ABB RAPID module: ANV4y1.mod

MODULE ANV4y1

	PERS tooldata Pen:=[TRUE,[[0,0,139],[1,0,0,0]],[0.5,[0,0,20],[1,0,0,0],0,0,0]];
	CONST robtarget origin :=[[0,0,0],[1,0,0,0],[0,0,-1,0],[9E+09,9E+09,9E+09,9E+09,9E+09,9E+09]];
	CONST robtarget home_1:=[[120,148.105008887,-250.933670218],[0.706940789,-0.015320621,0.015320621,0.706940789],[0,0,0,0],[9E+09,9E+09,9E+09,9E+09,9E+09,9E+09]];
	TASK PERS wobjdata paper_obj:=[FALSE,TRUE,"",[[1355,120,401],[0,-0.707106781,0.707106781,0]],[[0,0,0],[1,0,0,0]]];
	VAR num array_x{8510}:= [145,144,144,144,144,144,144,144,144,144,144,144,144,144,144,144,144,144,144,144,144,144,144,144,144,144,144,144,144,144,144,146,146,147,147,148,148,149,149,150,150,151,151,152,152,153,153,154,154,154,154,155,155,156,156,157,157,158,158,159,159,160,160,161,161,162,162,162,162,161,161,160,160,159,159,158,158,157,157,156,156,155,155,154,154,153,153,152,152,151,151,150,150,149,149,149,149,148,148,147,147,146,146,145,145,144,144,143,143,142,142,141,141,140,140,140,140,139,139,138,138,137,137,137,137,136,136,136,136,135,135,135,135,134,134,133,133,133,133,132,132,132,132,131,131,131,131,130,130,130,130,129,129,129,129,128,128,127,127,127,127,126,126,126,126,125,125,125,125,124,124,124,124,123,123,123,123,122,122,122,122,121,121,120,120,120,120,119,119,119,119,118,118,118,118,117,117,117,117,116,116,116,116,115,115,115,115,114,114,113,113,113,113,112,112,112,112,111,111,111,111,111,111,109,109,108,108,107,107,106,106,106,106,105,105,105,105,105,105,105,105,105,105,105,105,105,105,105,105,105,105,105,105,105,105,105,105,105,105,105,105,105,105,105,105,105,105,105,105,105,105,105,105,106,106,106,106,106,106,106,106,106,106,106,106,106,106,106,106,106,106,106,106,106,106,106,106,106,106,106,106,106,106,106,106,106,106,106,106,106,106,106,106,106,106,105,105,105,105,103,103,103,103,104,104,104,104,104,104,104,104,104,104,104,104,104,104,104,104,104,104,104,104,104,104,104,104,104,104,104,104,104,104,104,104,104,104,104,104,104,104,104,104,104,104,103,103,103,103,103,103,103,103,103,103,103,103,103,103,103,103,103,103,103,103,103,103,103,103,103,103,103,103,103,103,103,103,103,103,103,103,103,103,103,103,103,103,101,101,100,100,99,99,98,98,97,97,97,97,97,97,98,98,101,101,102,102,102,102,102,102,101,101,101,101,100,100,99,99,98,98,97,97,98,98,99,99,100,100,101,101,102,102,102,102,102,102,101,101,101,101,100,100,99,99,98,98,98,98,91,91,92,92,93,93,93,93,94,94,95,95,96,96,97,97,97,97,95,95,95,95,95,95,94,94,94,94,93,93,93,93,92,92,92,92,91,91,91,91,90,90,90,90,89,89,89,89,90,90,89,89,89,89,88,88,88,88,87,87,87,87,86,86,86,86,86,86,85,85,84,84,83,83,82,82,82,82,81,81,80,80,79,79,78,78,75,75,75,75,76,76,76,76,77,77,77,77,77,77,78,78,78,78,79,79,79,79,79,79,80,80,80,80,81,81,81,81,81,81,82,82,82,82,83,83,83,83,83,83,84,84,84,84,85,85,85,85,86,86,86,86,86,86,87,87,87,87,87,87,88,88,88,88,88,88,81,81,80,80,80,80,79,79,79,79,79,79,78,78,78,78,77,77,77,77,76,76,76,76,76,76,75,75,75,75,75,75,74,74,74,74,74,74,73,73,73,73,72,72,72,72,71,71,71,71,71,71,70,70,70,70,69,69,69,69,68,68,68,68,68,68,68,68,67,67,67,67,67,67,65,65,65,65,65,65,66,66,66,66,66,66,67,67,67,67,68,68,68,68,69,69,69,69,69,69,70,70,70,70,71,71,71,71,72,72,72,72,73,73,73,73,74,74,74,74,74,74,75,75,76,76,77,77,78,78,81,81,82,82,82,82,83,83,83,83,83,83,84,84,84,84,84,84,85,85,85,85,85,85,86,86,86,86,87,87,87,87,88,88,88,88,88,88,86,86,84,84,84,84,83,83,83,83,82,82,81,81,80,80,79,79,58,58,59,59,59,59,60,60,60,60,60,60,60,60,60,60,60,60,60,60,60,60,60,60,59,59,58,58,57,57,56,56,55,55,54,54,53,53,52,52,51,51,50,50,49,49,48,48,47,47,46,46,45,45,44,44,43,43,42,42,41,41,41,41,40,40,40,40,40,40,40,40,38,38,38,38,37,37,36,36,35,35,34,34,33,33,32,32,31,31,31,31,31,31,32,32,32,32,32,32,33,33,33,33,33,33,34,34,35,35,36,36,36,36,37,37,37,37,37,37,37,37,36,36,39,39,39,39,39,39,38,38,38,38,38,38,37,37,37,37,37,37,32,32,32,32,32,32,32,32,31,31,31,31,31,31,30,30,30,30,30,30,29,29,29,29,29,29,28,28,28,28,28,28,36,36,37,37,38,38,39,39,38,38,38,38,38,38,38,38,38,38,36,36,36,36,36,36,36,36,36,36,37,37,37,37,39,39,39,39,39,39,39,39,37,37,37,37,37,37,39,39,40,40,40,40,40,40,38,38,38,38,38,38,38,38,38,38,39,39,40,40,41,41,53,53,53,53,53,53,53,53,52,52,52,52,52,52,52,52,52,52,52,52,52,52,52,52,52,52,53,53,54,54,54,54,54,54,54,54,54,54,54,54,54,54,54,54,55,55,55,55,55,55,55,55,54,54,53,53,54,54,54,54,54,54,54,54,55,55,55,55,55,55,55,55,55,55,55,55,55,55,55,55,56,56,56,56,56,56,56,56,56,56,56,56,57,57,57,57,57,57,58,58,58,58,61,61,60,60,60,60,60,60,59,59,59,59,59,59,58,58,58,58,58,58,58,58,58,58,58,58,57,57,57,57,57,57,57,57,57,57,57,57,57,57,57,57,56,56,56,56,56,56,56,56,56,56,56,56,64,64,64,64,64,64,63,63,63,63,63,63,62,62,62,62,62,62,61,61,61,61,61,61,61,61,60,60,60,60,60,60,59,59,59,59,59,59,58,58,58,58,58,58,58,58,57,57,57,57,57,57,57,57,57,57,57,57,56,56,53,53,53,53,53,53,53,53,53,53,52,52,51,51,51,51,50,50,50,50,49,49,49,49,48,48,47,47,46,46,45,45,44,44,43,43,43,43,43,43,44,44,45,45,46,46,47,47,48,48,49,49,50,50,51,51,52,52,54,54,54,54,56,56,56,56,56,56,57,57,57,57,58,58,59,59,60,60,61,61,62,62,63,63,63,63,64,64,65,65,67,67,67,67,68,68,69,69,69,69,67,67,67,67,68,68,67,67,68,68,69,69,70,70,71,71,72,72,73,73,74,74,75,75,76,76,77,77,78,78,79,79,80,80,81,81,82,82,83,83,84,84,85,85,86,86,87,87,86,86,85,85,84,84,83,83,82,82,81,81,80,80,79,79,78,78,77,77,76,76,75,75,74,74,73,73,72,72,71,71,70,70,69,69,69,69,69,69,69,69,69,69,69,69,72,72,71,71,71,71,72,72,73,73,74,74,75,75,76,76,77,77,78,78,79,79,80,80,81,81,82,82,83,83,84,84,85,85,86,86,85,85,86,86,87,87,87,87,84,84,83,83,82,82,82,82,81,81,80,80,79,79,79,79,79,79,80,80,81,81,82,82,83,83,84,84,85,85,85,85,86,86,88,88,89,89,89,89,89,89,88,88,87,87,81,81,80,80,79,79,78,78,81,81,81,81,80,80,79,79,78,78,78,78,80,80,80,80,80,80,80,80,79,79,78,78,78,78,78,78,78,78,78,78,78,78,78,78,76,76,76,76,76,76,76,76,76,76,76,76,76,76,76,76,76,76,76,76,77,77,81,81,82,82,83,83,82,82,83,83,84,84,84,84,85,85,86,86,86,86,87,87,86,86,86,86,86,86,87,87,87,87,88,88,89,89,89,89,88,88,89,89,89,89,90,90,108,108,108,108,108,108,108,108,108,108,108,108,108,108,108,108,109,109,109,109,109,109,109,109,109,109,108,108,107,107,106,106,105,105,104,104,103,103,103,103,102,102,101,101,100,100,99,99,98,98,97,97,97,97,96,96,96,96,95,95,94,94,93,93,92,92,91,91,90,90,89,89,88,88,87,87,86,86,85,85,85,85,85,85,86,86,90,90,89,89,89,89,89,89,89,89,90,90,91,91,92,92,92,92,93,93,92,92,91,91,88,88,89,89,90,90,91,91,92,92,93,93,94,94,95,95,96,96,97,97,97,97,98,98,99,99,100,100,100,100,101,101,89,89,87,87,88,88,89,89,89,89,88,88,87,87,86,86,85,85,84,84,82,82,81,81,80,80,79,79,78,78,77,77,76,76,75,75,74,74,73,73,72,72,71,71,70,70,69,69,68,68,67,67,67,67,66,66,66,66,66,66,66,66,67,67,68,68,69,69,69,69,70,70,71,71,72,72,73,73,74,74,75,75,76,76,77,77,78,78,79,79,80,80,81,81,82,82,83,83,83,83,83,83,82,82,81,81,80,80,79,79,78,78,77,77,76,76,75,75,74,74,73,73,72,72,71,71,70,70,69,69,69,69,68,68,68,68,67,67,67,67,70,70,71,71,72,72,73,73,74,74,75,75,76,76,77,77,78,78,79,79,80,80,81,81,81,81,82,82,82,82,82,82,81,81,80,80,79,79,78,78,77,77,76,76,75,75,74,74,73,73,72,72,71,71,70,70,71,71,73,73,70,70,69,69,68,68,67,67,67,67,64,64,64,64,63,63,63,63,63,63,63,63,62,62,61,61,60,60,59,59,59,59,59,59,59,59,59,59,59,59,59,59,60,60,60,60,60,60,60,60,61,61,61,61,61,61,62,62,62,62,62,62,62,62,62,62,63,63,63,63,63,63,64,64,64,64,64,64,64,64,65,65,65,65,65,65,66,66,66,66,66,66,68,68,68,68,69,69,69,69,70,70,70,70,71,71,71,71,72,72,72,72,72,72,73,73,73,73,74,74,74,74,75,75,76,76,76,76,75,75,74,74,73,73,72,72,72,72,71,71,71,71,71,71,70,70,70,70,68,68,67,67,67,67,66,66,66,66,66,66,66,66,66,66,65,65,65,65,65,65,67,67,68,68,68,68,69,69,69,69,69,69,70,70,71,71,72,72,73,73,74,74,75,75,76,76,77,77,78,78,79,79,80,80,81,81,82,82,83,83,84,84,85,85,85,85,86,86,86,86,87,87,88,88,88,88,89,89,89,89,90,90,91,91,91,91,92,92,93,93,94,94,95,95,96,96,97,97,98,98,99,99,100,100,101,101,102,102,103,103,104,104,105,105,106,106,107,107,108,108,109,109,109,109,110,110,110,110,111,111,111,111,112,112,113,113,117,117,119,119,119,119,118,118,117,117,116,116,115,115,114,114,113,113,112,112,111,111,110,110,109,109,108,108,107,107,106,106,105,105,104,104,104,104,103,103,104,104,105,105,106,106,107,107,107,107,108,108,109,109,110,110,112,112,113,113,115,115,116,116,116,116,116,116,116,116,115,115,115,115,114,114,114,114,114,114,113,113,112,112,111,111,112,112,113,113,113,113,114,114,114,114,115,115,115,115,116,116,116,116,117,117,117,117,118,118,118,118,119,119,119,119,119,119,120,120,120,120,121,121,122,122,122,122,123,123,124,124,124,124,125,125,125,125,126,126,127,127,127,127,128,128,129,129,130,130,130,130,131,131,132,132,132,132,133,133,134,134,135,135,136,136,137,137,138,138,139,139,140,140,141,141,142,142,143,143,144,144,145,145,146,146,147,147,148,148,149,149,150,150,151,151,152,152,153,153,154,154,155,155,156,156,157,157,158,158,159,159,160,160,161,161,161,161,162,162,162,162,162,162,161,161,160,160,159,159,159,159,158,158,157,157,156,156,154,154,155,155,156,156,162,162,162,162,161,161,160,160,159,159,158,158,157,157,156,156,155,155,154,154,153,153,152,152,142,142,142,142,142,142,142,142,142,142,142,142,142,142,142,142,141,141,141,141,141,141,141,141,141,141,140,140,139,139,139,139,139,139,139,139,139,139,140,140,140,140,140,140,140,140,140,140,140,140,140,140,141,141,143,143,143,143,143,143,143,143,141,141,141,141,141,141,141,141,143,143,143,143,143,143,144,144,144,144,144,144,144,144,144,144,144,144,143,143,143,143,143,143,142,142,141,141,141,141,141,141,142,142,142,142,142,142,142,142,142,142,142,142,141,141,141,141,133,133,132,132,131,131,130,130,130,130,129,129,129,129,128,128,127,127,126,126,125,125,124,124,123,123,122,122,121,121,121,121,121,121,119,119,118,118,119,119,118,118,117,117,117,117,117,117,116,116,116,116,115,115,115,115,114,114,114,114,114,114,113,113,113,113,112,112,112,112,111,111,110,110,110,110,108,108,109,109,109,109,110,110,110,110,111,111,111,111,111,111,112,112,112,112,112,112,113,113,113,113,114,114,114,114,115,115,115,115,115,115,117,117,118,118,119,119,119,119,118,118,116,116,115,115,115,115,115,115,114,114,114,114,113,113,113,113,113,113,112,112,112,112,111,111,111,111,110,110,110,110,109,109,109,109,108,108,108,108,108,108,107,107,107,107,106,106,106,106,105,105,105,105,104,104,103,103,103,103,102,102,102,102,101,101,100,100,99,99,99,99,98,98,97,97,97,97,97,97,97,97,97,97,97,97,97,97,97,97,97,97,97,97,97,97,97,97,97,97,97,97,97,97,98,98,99,99,100,100,100,100,101,101,102,102,102,102,103,103,104,104,104,104,105,105,106,106,107,107,108,108,108,108,109,109,110,110,110,110,111,111,111,111,112,112,112,112,113,113,113,113,113,113,114,114,114,114,115,115,115,115,118,118,118,118,119,119,120,120,120,120,121,121,122,122,123,123,124,124,125,125,126,126,127,127,130,130,131,131,132,132,133,133,134,134,134,134,134,134,134,134,135,135,135,135,136,136,137,137,138,138,139,139,140,140,140,140,140,140,140,140,141,141,142,142,143,143,144,144,145,145,144,144,143,143,145,145,145,145,145,145,144,144,146,146,146,146,144,144,144,144,144,144,143,143,142,142,142,142,142,142,143,143,142,142,141,141,140,140,139,139,138,138,137,137,136,136,136,136,136,136,135,135,133,133,134,134,134,134,134,134,135,135,136,136,138,138,139,139,140,140,138,138,137,137,135,135,135,135,135,135,136,136,137,137,138,138,139,139,139,139,140,140,141,141,142,142,143,143,147,147,148,148,149,149,152,152,153,153,154,154,155,155,156,156,157,157,158,158,157,157,155,155,155,155,154,154,154,154,152,152,152,152,151,151,151,151,150,150,149,149,150,150,149,149,148,148,148,148,148,148,148,148,149,149,150,150,150,150,150,150,151,151,151,151,151,151,147,147,146,146,146,146,146,146,146,146,146,146,147,147,147,147,148,148,149,149,150,150,151,151,152,152,152,152,153,153,153,153,153,153,152,152,153,153,153,153,154,154,155,155,156,156,157,157,157,157,158,158,159,159,160,160,161,161,161,161,162,162,162,162,161,161,160,160,159,159,158,158,157,157,156,156,155,155,155,155,154,154,152,152,153,153,153,153,153,153,152,152,154,154,155,155,156,156,157,157,157,157,157,157,156,156,158,158,158,158,159,159,158,158,159,159,159,159,159,159,159,159,160,160,160,160,160,160,159,159,158,158,157,157,156,156,155,155,154,154,153,153,152,152,151,151,150,150,150,150,149,149,148,148,147,147,146,146,146,146,145,145,144,144,143,143,142,142,141,141,140,140,139,139,138,138,137,137,136,136,135,135,134,134,133,133,133,133,133,133,133,133,132,132,131,131,131,131,130,130,130,130,130,130,131,131,131,131,131,131,130,130,130,130,130,130,129,129,128,128,127,127,126,126,125,125,124,124,123,123,122,122,121,121,120,120,119,119,118,118,117,117,116,116,115,115,114,114,113,113,113,113,112,112,112,112,112,112,111,111,111,111,111,111,111,111,111,111,111,111,110,110,110,110,110,110,111,111,112,112,113,113,114,114,114,114,115,115,115,115,115,115,113,113,113,113,113,113,115,115,115,115,114,114,114,114,113,113,112,112,112,112,112,112,111,111,110,110,109,109,109,109,108,108,109,109,109,109,110,110,110,110,112,112,112,112,111,111,110,110,110,110,110,110,108,108,107,107,107,107,107,107,106,106,105,105,104,104,103,103,102,102,101,101,100,100,99,99,98,98,97,97,96,96,95,95,94,94,93,93,92,92,91,91,90,90,89,89,88,88,87,87,86,86,86,86,85,85,84,84,83,83,82,82,82,82,81,81,80,80,80,80,79,79,79,79,78,78,77,77,76,76,76,76,75,75,74,74,73,73,72,72,71,71,70,70,69,69,69,69,68,68,68,68,67,67,67,67,67,67,69,69,66,66,66,66,66,66,66,66,66,66,65,65,66,66,67,67,68,68,69,69,70,70,71,71,71,71,70,70,70,70,70,70,69,69,68,68,67,67,67,67,67,67,67,67,68,68,69,69,70,70,69,69,68,68,67,67,66,66,65,65,65,65,64,64,64,64,63,63,63,63,63,63,63,63,63,63,64,64,64,64,64,64,65,65,65,65,65,65,65,65,66,66,67,67,68,68,69,69,70,70,71,71,71,71,72,72,70,70,69,69,68,68,67,67,66,66,57,57,56,56,56,56,55,55,55,55,54,54,53,53,52,52,51,51,50,50,49,49,48,48,47,47,46,46,44,44,43,43,42,42,41,41,40,40,39,39,39,39,40,40,41,41,42,42,43,43,44,44,45,45,46,46,47,47,48,48,49,49,50,50,51,51,52,52,53,53,54,54,54,54,55,55,56,56,57,57,58,58,59,59,60,60,61,61,62,62,63,63,64,64,65,65,66,66,67,67,68,68,68,68,67,67,67,67,66,66,65,65,65,65,64,64,63,63,62,62,61,61,60,60,59,59,58,58,57,57,56,56,55,55,54,54,53,53,52,52,51,51,50,50,49,49,49,49,48,48,47,47,46,46,45,45,44,44,43,43,43,43,42,42,41,41,41,41,40,40,39,39,39,39,38,38,38,38,39,39,40,40,40,40,41,41,42,42,43,43,44,44,45,45,46,46,47,47,48,48,49,49,50,50,50,50,50,50,49,49,48,48,47,47,46,46,45,45,44,44,43,43,42,42,41,41,40,40,39,39,37,37,37,37,37,37,37,37,36,36,35,35,34,34,34,34,33,33,32,32,32,32,31,31,31,31,30,30,30,30,29,29,29,29,28,28,28,28,27,27,27,27,27,27,26,26,24,24,26,26,26,26,26,26,26,26,26,26,26,26,26,26,26,26,27,27,27,27,28,28,28,28,28,28,29,29,29,29,30,30,30,30,31,31,32,32,34,34,35,35,36,36,37,37,38,38,39,39,40,40,40,40,40,40,39,39,38,38,37,37,36,36,35,35,34,34,36,36,36,36,36,36,35,35,34,34,33,33,33,33,33,33,33,33,34,34,35,35,36,36,45,45,46,46,46,46,45,45,45,45,44,44,44,44,44,44,44,44,44,44,45,45,46,46,46,46,46,46,46,46,47,47,47,47,47,47,48,48,48,48,48,48,47,47,46,46,46,46,45,45,47,47,46,46,45,45,44,44,43,43,42,42,41,41,40,40,39,39,38,38,38,38,38,38,39,39,40,40,41,41,42,42,43,43,44,44,45,45,46,46,47,47,48,48,49,49,48,48,49,49,50,50,50,50,50,50,57,57,58,58,58,58,58,58,58,58,57,57,57,57,56,56,56,56,55,55,55,55,54,54,54,54,53,53,52,52,51,51,51,51,50,50,50,50,50,50,51,51,51,51,52,52,54,54,55,55,55,55,52,52,52,52,52,52,51,51,50,50,49,49,48,48,47,47,47,47,47,47,49,49,50,50,51,51,52,52,52,52,52,52,51,51,51,51,50,50,50,50,49,49,49,49,55,55,55,55,55,55,55,55,55,55,55,55,55,55,55,55,56,56,56,56,56,56,56,56,57,57,57,57,58,58,59,59,60,60,60,60,59,59,59,59,58,58,58,58,58,58,58,58,57,57,57,57,57,57,57,57,57,57,57,57,57,57,57,57,59,59,59,59,59,59,59,59,59,59,59,59,59,59,61,61,61,61,61,61,61,61,60,60,63,63,63,63,62,62,62,62,61,61,66,66,69,69,70,70,74,74,75,75,76,76,77,77,78,78,79,79,80,80,81,81,82,82,82,82,83,83,84,84,85,85,85,85,86,86,87,87,88,88,89,89,90,90,91,91,91,91,91,91,90,90,89,89,89,89,88,88,88,88,87,87,87,87,86,86,85,85,84,84,83,83,82,82,81,81,80,80,74,74,75,75,76,76,77,77,77,77,77,77,79,79,80,80,81,81,82,82,83,83,84,84,85,85,85,85,87,87,88,88,89,89,90,90,91,91,93,93,94,94,95,95,96,96,97,97,98,98,99,99,100,100,101,101,102,102,106,106,105,105,104,104,103,103,101,101,100,100,97,97,96,96,95,95,94,94,95,95,93,93,91,91,92,92,93,93,94,94,92,92,91,91,87,87,87,87,87,87,84,84,85,85,86,86,87,87,88,88,89,89,90,90,91,91,92,92,93,93,93,93,94,94,94,94,95,95,95,95,96,96,96,96,97,97,97,97,98,98,98,98,99,99,100,100,101,101,101,101,101,101,100,100,100,100,99,99,98,98,97,97,96,96,98,98,99,99,100,100,101,101,102,102,102,102,103,103,103,103,103,103,104,104,104,104,105,105,105,105,106,106,106,106,107,107,107,107,107,107,108,108,109,109,109,109,111,111,114,114,113,113,114,114,114,114,114,114,113,113,113,113,113,113,112,112,112,112,111,111,111,111,110,110,110,110,109,109,109,109,108,108,108,108,108,108,107,107,107,107,106,106,106,106,105,105,105,105,104,104,103,103,103,103,102,102,102,102,101,101,100,100,99,99,98,98,97,97,96,96,95,95,94,94,93,93,92,92,91,91,90,90,89,89,88,88,87,87,86,86,85,85,84,84,83,83,82,82,81,81,80,80,79,79,78,78,77,77,76,76,75,75,74,74,73,73,72,72,71,71,70,70,69,69,68,68,67,67,66,66,65,65,65,65,64,64,63,63,63,63,62,62,62,62,61,61,61,61,60,60,60,60,59,59,59,59,58,58,58,58,57,57,57,57,56,56,55,55,54,54,53,53,52,52,51,51,50,50,49,49,48,48,47,47,46,46,45,45,44,44,43,43,42,42,41,41,40,40,39,39,39,39,40,40,42,42,44,44,46,46,47,47,48,48,47,47,46,46,45,45,44,44,43,43,41,41,40,40,40,40,39,39,38,38,38,38,37,37,37,37,36,36,36,36,35,35,35,35,34,34,34,34,34,34,33,33,33,33,32,32,32,32,32,32,29,29,23,23,22,22,18,18,19,19,20,20,21,21,23,23,22,22,21,21,20,20,19,19,18,18,16,16,15,15,14,14,14,14,15,15,16,16,17,17,15,15,16,16,16,16,17,17,17,17,18,18,18,18,18,18,19,19,19,19,19,19,19,19,19,19,19,19,19,19,20,20,20,20,22,22,22,22,21,21,21,21,21,21,21,21,21,21,21,21,21,21,20,20,20,20,20,20,19,19,26,26,26,26,26,26,26,26,27,27,27,27,28,28,28,28,28,28,28,28,28,28,28,28,27,27,27,27,28,28,28,28,28,28,28,28,28,28,30,30,30,30,30,30,30,30,30,30,29,29,30,30,31,31,30,30,31,31,32,32,33,33,34,34,33,33,33,33,33,33,33,33,32,32,31,31,30,30,31,31,31,31,31,31,30,30,29,29,28,28,29,29,29,29,27,27,27,27,28,28,28,28,29,29,29,29,30,30,30,30,32,32,32,32,33,33,34,34,36,36,36,36,35,35,35,35,35,35,36,36,36,36,35,35,37,37,36,36,35,35,34,34,33,33,32,32,33,33,34,34,35,35,36,36,37,37,38,38,39,39,39,39,40,40,41,41,40,40,44,44,45,45,46,46,47,47,47,47,47,47,43,43,43,43,43,43,43,43,43,43,43,43,44,44,45,45,46,46,45,45,45,45,45,45,47,47,47,47,47,47,47,47,46,46,46,46,46,46,46,46,45,45,45,45,45,45,45,45,45,45,44,44,44,44,44,44,44,44,44,44,43,43,43,43,43,43,43,43,42,42,42,42,42,42,42,42,42,42,41,41,41,41,41,41,39,39,39,39,39,39,39,39,40,40,40,40,40,40,40,40,41,41,41,41,41,41,41,41,41,41,42,42,42,42,42,42,42,42,42,42,43,43,43,43,43,43,44,44,44,44,44,44,44,44,42,42,42,42,42,42,42,42,42,42,40,40,40,40,40,40,40,40,40,40,40,40,39,39,38,38,37,37,36,36,35,35,34,34,33,33,32,32,31,31,30,30,29,29,29,29,29,29,29,29,29,29,29,29,27,27,27,27,27,27,27,27,28,28,29,29,30,30,31,31,32,32,33,33,34,34,35,35,36,36,37,37,38,38,39,39,40,40,27,27,25,25,25,25,25,25,25,25,25,25,25,25,25,25,26,26,26,26,26,26,26,26,26,26,26,26,26,26,26,26,26,26,26,26,26,26,26,26,26,26,26,26,26,26,27,27,27,27,27,27,27,27,14,14,14,14,14,14,13,13,13,13,13,13,13,13,12,12,12,12,12,12,11,11,11,11,11,11,11,11,11,11,10,10,10,10,10,10,10,10,10,10,10,10,9,9,9,9,9,9,9,9,8,8,8,8,8,8,8,8,8,8,8,8,8,8,8,8,8,8,8,8,8,8,25,25,25,25,24,24,24,24,24,24,24,24,24,24,24,24,24,24,24,24,24,24,24,24,24,24,24,24,24,24,24,24,24,24,24,24,24,24,24,24,24,24,25,25,25,25,25,25,25,25,25,25,25,25,25,25,25,25,25,25,25,25,25,25,25,25,24,24,24,24,23,23,23,23,23,23,22,22,22,22,21,21,20,20,19,19,18,18,17,17,16,16,15,15,14,14,13,13,12,12,11,11,11,11,10,10,10,10,9,9,8,8,8,8,8,8,7,7,7,7,7,7,7,7,7,7,6,6,6,6,6,6,6,6,6,6,6,6,6,6,6,6,6,6,6,6,6,6,6,6,6,6,6,6,5,5,5,5,5,5,5,5,5,5,5,5,5,5,5,5,5,5,5,5,5,5,5,5,5,5,5,5,5,5,5,5,5,5,5,5,5,5,5,5,6,6,6,6,6,6,6,6,6,6,6,6,6,6,6,6,6,6,7,7,7,7,7,7,7,7,7,7,7,7,8,8,8,8,8,8,8,8,8,8,8,8,9,9,9,9,9,9,9,9,9,9,9,9,10,10,10,10,10,10,10,10,11,11,11,11,11,11,11,11,12,12,12,12,12,12,13,13,13,13,13,13,11,11,11,11,10,10,10,10,10,10,9,9,9,9,9,9,9,9,8,8,8,8,8,8,8,8,7,7,7,7,7,7,7,7,7,7,6,6,6,6,6,6,6,6,6,6,6,6,5,5,5,5,5,5,5,5,5,5,5,5,5,5,4,4,4,4,4,4,4,4,4,4,4,4,4,4,4,4,4,4,3,3,3,3,3,3,3,3,3,3,3,3,3,3,3,3,3,3,3,3,3,3,3,3,3,3,3,3,3,3,3,3,3,3,2,2,1,1,3,3,1,1,1,1,1,1,1,1,1,1,1,1,1,1,1,1,2,2,2,2,2,2,2,2,2,2,3,3,3,3,3,3,4,4,4,4,4,4,5,5,5,5,5,5,6,6,6,6,6,6,7,7,7,7,7,7,8,8,8,8,9,9,9,9,9,9,10,10,10,10,11,11,11,11,11,11,12,12,12,12,13,13,13,13,13,13,14,14,14,14,14,14,15,15,15,15,15,15,16,16,16,16,16,16,17,17,17,17,18,18,18,18,19,19,19,19,20,20,20,20,20,20,21,21,21,21,21,21,22,22,22,22,23,23,23,23,23,23,24,24,24,24,25,25,25,25,26,26,26,26,27,27,27,27,28,28,28,28,29,29,30,30,31,31,32,32,33,33,34,34,35,35,36,36,37,37,38,38,22,22,21,21,20,20,19,19,18,18,18,18,17,17,17,17,16,16,15,15,15,15,14,14,14,14,13,13,13,13,12,12,11,11,11,11,10,10,10,10,9,9,9,9,8,8,8,8,7,7,7,7,6,6,6,6,6,6,5,5,5,5,5,5,5,5,6,6,6,6,7,7,7,7,8,8,9,9,7,7,6,6,5,5,4,4,2,2,3,3,3,3,4,4,4,4,5,5,5,5,5,5,6,6,6,6,7,7,7,7,8,8,8,8,9,9,9,9,10,10,10,10,11,11,12,12,13,13,14,14,15,15,16,16,16,16,16,16,16,16,17,17,17,17,17,17,17,17,18,18,17,17,16,16,15,15,14,14,13,13,12,12,12,12,10,10,7,7,8,8,9,9,10,10,11,11,12,12,13,13,10,10,11,11,12,12,13,13,14,14,15,15,16,16,20,20,20,20,20,20,20,20,20,20,21,21,21,21,21,21,21,21,22,22,22,22,23,23,24,24,25,25,26,26,27,27,27,27,28,28,28,28,26,26,25,25,24,24,21,21,22,22,23,23,24,24,24,24,26,26,27,27,27,27,28,28,30,30,30,30,30,30,31,31,31,31,32,32,33,33,34,34,35,35,35,35,35,35,35,35,34,34,34,34,34,34,37,37,37,37,37,37,37,37,38,38,38,38,38,38,39,39,40,40,41,41,42,42,43,43,43,43,44,44,44,44,44,44,45,45,45,45,47,47,47,47,47,47,48,48,49,49,50,50,51,51,52,52,51,51,51,51,51,51,51,51,53,53,54,54,54,54,54,54,54,54,55,55,56,56,57,57,58,58,59,59,59,59,59,59,59,59,68,68,68,68,69,69,72,72,73,73,73,73,74,74,74,74,74,74,75,75,75,75,71,71,70,70,69,69,69,69,70,70,71,71,72,72,73,73,74,74,76,76,77,77,78,78,79,79,80,80,81,81,82,82,83,83,84,84,85,85,86,86,87,87,89,89,89,89,89,89,90,90,91,91,92,92,93,93,94,94,95,95,96,96,97,97,98,98,99,99,96,96,94,94,94,94,89,89,88,88,88,88,88,88,88,88,92,92,93,93,94,94,94,94,98,98,99,99,99,99,99,99,100,100,100,100,101,101,101,101,101,101,101,101,100,100,103,103,104,104,105,105,106,106,107,107,108,108,109,109,110,110,111,111,112,112,113,113,113,113,114,114,110,110,109,109,108,108,108,108,111,111,112,112,113,113,117,117,118,118,118,118,119,119,119,119,120,120,120,120,121,121,121,121,122,122,123,123,124,124,125,125,126,126,127,127,127,127,127,127,127,127,128,128,128,128,128,128,128,128,129,129,128,128,127,127,126,126,125,125,124,124,124,124,123,123,122,122,121,121,120,120,119,119,117,117,118,118,118,118,121,121,123,123,123,123,122,122,121,121,117,117,116,116,116,116,115,115,115,115,115,115,114,114,116,116,115,115,114,114,113,113,111,111,110,110,109,109,108,108,107,107,112,112,112,112,113,113,113,113,113,113,112,112,111,111,110,110,109,109,108,108,103,103,103,103,103,103,103,103,104,104,105,105,106,106,107,107,108,108,108,108,108,108,107,107,106,106,106,106,105,105,104,104,103,103,105,105,104,104,103,103,101,101,102,102,102,102,102,102,101,101,99,99,99,99,98,98,97,97,96,96,95,95,95,95,94,94,92,92,92,92,92,92,91,91,90,90,89,89,88,88,87,87,85,85,85,85,84,84,85,85,85,85,84,84,83,83,82,82,83,83,82,82,81,81,80,80,80,80,81,81,80,80,79,79,78,78,77,77,76,76,75,75,75,75,75,75,75,75,76,76,80,80,81,81,82,82,83,83,84,84,85,85,85,85,83,83,82,82,81,81,81,81,84,84,85,85,86,86,86,86,85,85,84,84,83,83,82,82,81,81,77,77,77,77,76,76,76,76,72,72,71,71,71,71,70,70,70,70,70,70,69,69,69,69,68,68,67,67,66,66,65,65,64,64,63,63,63,63,62,62,62,62,62,62,62,62,62,62,66,66,66,66,66,66,66,66,66,66,66,66,65,65,64,64,63,63,62,62,61,61,61,61,61,61,61,61,59,59,58,58,58,58,58,58,53,53,53,53,53,53,57,57,57,57,57,57,56,56,55,55,54,54,53,53,52,52,50,50,50,50,47,47,50,50,50,50,49,49,48,48,47,47,46,46,45,45,44,44,44,44,43,43,43,43,43,43,41,41,41,41,41,41,41,41,40,40,39,39,38,38,37,37,36,36,36,36,36,36,36,36,34,34,33,33,33,33,33,33,32,32,31,31,30,30,29,29,28,28,28,28,27,27,26,26,25,25,24,24,23,23,22,22,22,22,21,21,19,19,18,18,18,18,17,17,16,16,15,15,14,14,13,13,12,12,11,11,10,10,10,10,9,9,8,8,7,7,7,7,7,7,10,10,13,13,14,14,15,15,17,17,18,18,19,19,20,20,21,21,23,23,22,22,23,23,23,23,24,24,24,24,25,25,26,26,26,26,27,27,27,27,28,28,28,28,29,29,29,29,30,30,30,30,31,31,31,31,29,29,28,28,27,27,26,26,22,22,21,21,20,20,21,21,22,22,25,25,24,24,25,25,26,26,27,27,28,28,29,29,28,28,29,29,32,32,32,32,32,32,31,31,30,30,29,29,30,30,31,31,32,32,32,32,33,33,33,33,34,34,34,34,34,34,35,35,35,35,34,34,34,34,33,33,33,33,32,32,32,32,39,39,40,40,40,40,41,41,41,41,42,42,42,42,43,43,44,44,45,45,46,46,47,47,48,48,49,49,49,49,49,49,49,49,49,49,49,49,44,44,45,45,44,44,43,43,42,42,42,42,39,39,38,38,38,38,37,37,37,37,37,37,38,38,39,39,40,40,41,41,42,42,43,43,44,44,45,45,46,46,47,47,48,48,49,49,50,50,57,57,57,57,57,57,58,58,59,59,60,60,61,61,62,62,62,62,64,64,65,65,67,67,68,68,69,69,70,70,66,66,65,65,64,64,63,63,62,62,58,58,58,58,59,59,59,59,59,59,60,60,59,59,59,59,59,59,60,60,61,61,62,62,63,63,64,64,64,64,64,64,65,65,65,65,66,66,66,66,67,67,67,67,68,68,68,68,69,69,69,69,70,70,72,72,73,73,74,74,75,75,76,76,77,77,78,78,79,79,80,80,81,81,81,81,81,81,80,80,79,79,78,78,77,77,76,76,76,76,76,76,77,77,78,78,79,79,80,80,80,80,80,80,80,80,79,79,78,78,77,77,76,76,75,75,75,75,72,72,72,72,71,71,71,71,71,71,71,71,70,70,70,70,70,70,71,71,72,72,73,73,74,74,75,75,76,76,77,77,78,78,79,79,80,80,80,80,81,81,81,81,82,82,82,82,83,83,83,83,84,84,84,84,85,85,85,85,85,85,86,86,86,86,87,87,87,87,88,88,88,88,89,89,90,90,91,91,92,92,93,93,94,94,95,95,95,95,95,95,95,95,91,91,91,91,90,90,89,89,89,89,90,90,83,83,84,84,85,85,86,86,87,87,88,88,89,89,90,90,91,91,92,92,93,93,94,94,95,95,96,96,96,96,96,96,96,96,96,96,98,98,99,99,100,100,101,101,102,102,103,103,103,103,103,103,103,103,99,99,99,99,99,99,99,99,100,100,100,100,100,100,100,100,101,101,102,102,103,103,104,104,105,105,106,106,107,107,108,108,107,107,106,106,105,105,105,105,105,105,105,105,106,106,107,107,108,108,109,109,110,110,110,110,110,110,109,109,109,109,109,109,110,110,111,111,111,111,112,112,112,112,112,112,111,111,109,109,110,110,111,111,115,115,116,116,117,117,118,118,119,119,120,120,121,121,122,122,123,123,124,124,121,121,120,120,120,120,119,119,115,115,114,114,114,114,114,114,114,114,115,115,115,115,116,116,117,117,118,118,118,118,117,117,116,116,115,115,114,114,113,113,113,113,113,113,114,114,115,115,116,116,117,117,118,118,119,119,120,120,121,121,122,122,123,123,123,123,124,124,124,124,124,124,124,124,123,123,123,123,122,122,121,121,122,122,123,123,124,124,124,124,125,125,129,129,130,130,130,130,130,130,131,131,131,131,132,132,132,132,133,133,133,133,134,134,134,134,135,135,136,136,136,136,137,137,137,137,138,138,138,138,139,139,139,139,140,140,141,141,141,141,142,142,142,142,143,143,144,144,145,145,145,145,146,146,146,146,147,147,148,148,148,148,149,149,149,149,150,150,150,150,151,151,152,152,152,152,153,153,153,153,154,154,154,154,155,155,155,155,153,153,152,152,150,150,149,149,148,148,147,147,146,146,144,144,143,143,142,142,141,141,141,141,140,140,139,139,139,139,138,138,137,137,136,136,145,145,146,146,148,148,149,149,150,150,151,151,152,152,153,153,153,153,155,155,156,156,157,157,157,157,157,157,158,158,157,157,156,156,156,156,157,157,158,158,158,158,159,159,159,159,159,159,159,159,158,158,158,158,157,157,157,157,156,156,155,155,155,155,154,154,153,153,152,152,151,151,150,150,149,149,148,148,147,147,146,146,146,146,145,145,145,145,144,144,143,143,142,142,141,141,140,140,139,139,138,138,137,137,136,136,135,135,134,134,133,133,132,132,131,131,131,131,129,129,128,128,128,128,128,128,128,128,129,129,129,129,130,130,130,130,131,131,132,132,133,133,134,134,135,135,136,136,137,137,138,138,139,139,140,140,141,141,142,142,143,143,143,143,142,142,141,141,140,140,139,139,138,138,138,138,137,137,137,137,136,136,135,135,135,135,135,135,135,135,134,134,133,133,132,132,131,131,131,131,131,131,131,131,131,131,131,131,132,132,132,132,132,132,133,133,133,133,134,134,135,135,136,136,137,137,138,138,137,137,137,137,139,139,139,139,140,140,141,141,142,142,143,143,144,144,144,144,143,143,143,143,142,142,141,141,142,142,142,142,142,142,144,144,144,144,146,146,146,146,146,146,147,147,148,148,149,149,150,150,151,151,151,151,154,154,155,155,156,156,157,157,158,158,155,155,154,154,153,153,152,152,147,147,147,147,148,148,148,148,148,148,149,149,149,149,149,149,149,149,148,148,149,149,150,150,151,151,152,152,153,153,153,153,153,153,154,154,154,154,154,154,155,155,156,156,156,156,157,157,157,157,158,158,158,158,159,159,159,159,160,160,160];
	VAR num array_y{8510}:= [209,208,208,207,207,206,206,205,205,204,204,203,203,202,202,201,201,200,200,199,199,198,198,197,197,196,196,195,195,194,194,195,195,195,195,195,195,196,196,196,196,196,196,196,196,196,196,196,196,197,197,197,197,197,197,197,197,197,197,197,197,197,197,197,197,197,197,195,195,195,195,195,195,195,195,195,195,195,195,195,195,195,195,194,194,194,194,194,194,194,194,194,194,194,194,193,193,193,193,193,193,193,193,192,192,192,192,192,192,192,192,191,191,191,191,190,190,190,190,189,189,189,189,188,188,188,188,187,187,187,187,186,186,186,186,186,186,185,185,185,185,184,184,184,184,183,183,183,183,182,182,182,182,181,181,181,181,181,181,180,180,180,180,179,179,179,179,178,178,178,178,177,177,177,177,176,176,176,176,175,175,175,175,175,175,174,174,174,174,173,173,173,173,172,172,172,172,171,171,171,171,170,170,170,170,169,169,169,169,169,169,168,168,168,168,167,167,167,167,166,166,165,165,165,165,166,166,166,166,165,165,166,166,166,166,167,167,168,168,169,169,170,170,171,171,172,172,173,173,174,174,175,175,176,176,177,177,178,178,179,179,180,180,181,181,182,182,183,183,184,184,185,185,187,187,188,188,189,189,190,190,191,191,192,192,193,193,194,194,195,195,196,196,197,197,198,198,199,199,200,200,201,201,202,202,203,203,204,204,205,205,206,206,207,207,208,208,209,209,209,209,208,208,207,207,206,206,205,205,204,204,203,203,202,202,201,201,200,200,199,199,198,198,197,197,196,196,195,195,194,194,193,193,192,192,191,191,190,190,189,189,188,188,187,187,186,186,185,185,184,184,183,183,182,182,181,181,180,180,179,179,178,178,177,177,176,176,175,175,174,174,173,173,172,172,171,171,170,170,169,169,167,167,166,166,165,165,166,166,166,166,166,166,167,167,167,167,168,168,169,169,169,169,167,167,167,167,168,168,169,169,169,169,170,170,170,170,170,170,170,170,189,189,188,188,188,188,188,188,188,188,188,188,189,189,190,190,190,190,191,191,191,191,191,191,191,191,190,190,195,195,197,197,199,199,200,200,201,201,203,203,205,205,207,207,209,209,209,209,208,208,207,207,206,206,205,205,204,204,203,203,202,202,201,201,200,200,199,199,198,198,197,197,196,196,195,195,193,193,192,192,191,191,190,190,189,189,188,188,187,187,187,187,186,186,185,185,184,184,182,182,180,180,179,179,178,178,177,177,175,175,173,173,172,172,171,171,172,172,172,172,173,173,173,173,174,174,175,175,175,175,176,176,177,177,178,178,179,179,179,179,180,180,180,180,181,181,182,182,182,182,183,183,184,184,185,185,186,186,186,186,187,187,188,188,189,189,189,189,190,190,191,191,191,191,192,192,193,193,193,193,194,194,195,195,195,195,194,194,193,193,192,192,191,191,190,190,190,190,189,189,188,188,187,187,186,186,185,185,184,184,184,184,183,183,182,182,182,182,181,181,180,180,180,180,179,179,178,178,177,177,176,176,175,175,174,174,174,174,173,173,172,172,171,171,170,170,169,169,168,168,167,167,167,167,166,166,165,165,166,166,167,167,168,168,168,168,169,169,170,170,171,171,172,172,174,174,175,175,175,175,176,176,177,177,178,178,179,179,180,180,181,181,182,182,183,183,184,184,185,185,185,185,186,186,187,187,188,188,190,190,192,192,194,194,196,196,197,197,198,198,198,198,199,199,200,200,200,200,201,201,202,202,202,202,203,203,204,204,204,204,205,205,206,206,207,207,207,207,208,208,209,209,209,209,206,206,205,205,204,204,203,203,202,202,200,200,198,198,196,196,209,209,208,208,207,207,206,206,205,205,204,204,203,203,202,202,201,201,200,200,199,199,198,198,198,198,198,198,198,198,197,197,197,197,197,197,197,197,197,197,197,197,196,196,196,196,196,196,196,196,195,195,195,195,195,195,194,194,194,194,194,194,195,195,196,196,197,197,198,198,199,199,199,199,198,198,198,198,198,198,198,198,198,198,198,198,198,198,198,198,199,199,200,200,200,200,201,201,202,202,203,203,204,204,205,205,205,205,205,205,205,205,204,204,203,203,202,202,201,201,200,200,200,200,201,201,202,202,203,203,204,204,205,205,206,206,207,207,208,208,209,209,209,209,208,208,207,207,206,206,205,205,204,204,203,203,203,203,202,202,201,201,200,200,199,199,198,198,197,197,196,196,195,195,192,192,193,193,193,193,191,191,191,191,190,190,189,189,188,188,187,187,191,191,190,190,189,189,188,188,187,187,186,186,185,185,186,186,185,185,184,184,183,183,184,184,183,183,182,182,182,182,181,181,180,180,179,179,181,181,180,180,179,179,178,178,177,177,177,177,178,178,177,177,171,171,170,170,169,169,168,168,167,167,166,166,165,165,164,164,163,163,162,162,161,161,160,160,159,159,159,159,159,159,160,160,161,161,162,162,163,163,164,164,165,165,166,166,168,168,169,169,170,170,171,171,172,172,172,172,173,173,174,174,175,175,176,176,177,177,178,178,179,179,180,180,181,181,182,182,183,183,184,184,185,185,186,186,187,187,188,188,189,189,190,190,191,191,192,192,193,193,194,194,195,195,195,195,195,195,194,194,193,193,193,193,192,192,191,191,190,190,189,189,188,188,187,187,186,186,185,185,184,184,183,183,182,182,181,181,180,180,179,179,178,178,177,177,176,176,175,175,174,174,173,173,172,172,171,171,165,165,164,164,163,163,162,162,161,161,160,160,159,159,158,158,157,157,156,156,155,155,154,154,153,153,152,152,151,151,150,150,149,149,148,148,147,147,145,145,144,144,143,143,142,142,141,141,140,140,139,139,138,138,137,137,136,136,134,134,132,132,133,133,134,134,135,135,136,136,137,137,137,137,138,138,138,138,139,139,139,139,140,140,140,140,140,140,139,139,138,138,137,137,137,137,136,136,135,135,135,135,134,134,134,134,134,134,133,133,133,133,132,132,132,132,131,131,131,131,130,130,129,129,130,130,131,131,132,132,134,134,134,134,133,133,132,132,132,132,132,132,132,132,131,131,131,131,131,131,129,129,130,130,130,130,130,130,129,129,128,128,127,127,127,127,126,126,125,125,127,127,128,128,128,128,128,128,129,129,129,129,129,129,129,129,130,130,130,130,130,130,131,131,131,131,131,131,131,131,132,132,132,132,132,132,129,129,129,129,128,128,128,128,128,128,128,128,127,127,127,127,127,127,127,127,126,126,126,126,126,126,126,126,126,126,125,125,125,125,125,125,125,125,123,123,122,122,121,121,120,120,119,119,116,116,116,116,115,115,114,114,114,114,114,114,114,114,114,114,114,114,114,114,114,114,114,114,114,114,114,114,114,114,114,114,114,114,114,114,112,112,111,111,111,111,110,110,111,111,111,111,111,111,112,112,112,112,112,112,112,112,111,111,110,110,110,110,110,110,109,109,109,109,109,109,109,109,108,108,108,108,109,109,109,109,108,108,107,107,107,107,107,107,103,103,103,103,103,103,103,103,102,102,101,101,101,101,101,101,101,101,100,100,99,99,98,98,97,97,96,96,96,96,93,93,94,94,95,95,96,96,97,97,98,98,99,99,101,101,100,100,99,99,98,98,97,97,96,96,95,95,94,94,93,93,92,92,92,92,88,88,87,87,87,87,89,89,89,89,89,89,88,88,88,88,88,88,87,87,91,91,92,92,93,93,94,94,94,94,95,95,95,95,95,95,94,94,91,91,91,91,92,92,93,93,94,94,95,95,96,96,97,97,98,98,99,99,100,100,101,101,102,102,103,103,104,104,105,105,106,106,107,107,108,108,109,109,110,110,111,111,111,111,112,112,112,112,113,113,113,113,114,114,114,114,114,114,115,115,116,116,115,115,115,115,115,115,114,114,114,114,114,114,114,114,114,114,114,114,114,114,118,118,118,118,119,119,120,120,120,120,120,120,120,120,119,119,118,118,117,117,117,117,117,117,117,117,118,118,119,119,120,120,121,121,129,129,130,130,130,130,130,130,131,131,131,131,132,132,132,132,133,133,133,133,134,134,134,134,135,135,135,135,136,136,137,137,136,136,135,135,135,135,135,135,134,134,133,133,133,133,134,134,134,134,134,134,133,133,133,133,133,133,132,132,132,132,132,132,131,131,132,132,132,132,133,133,133,133,133,133,133,133,133,133,134,134,134,134,135,135,135,135,136,136,137,137,138,138,138,138,138,138,138,138,137,137,137,137,137,137,136,136,136,136,136,136,136,136,136,136,136,136,136,136,137,137,137,137,137,137,138,138,138,138,139,139,140,140,141,141,140,140,140,140,140,140,140,140,140,140,139,139,139,139,139,139,139,139,139,139,139,139,140,140,140,140,141,141,141,141,142,142,142,142,143,143,144,144,144,144,143,143,143,143,143,143,143,143,144,144,144,144,144,144,144,144,145,145,145,145,146,146,146,146,147,147,148,148,148,148,149,149,149,149,149,149,149,149,149,149,149,149,149,149,149,149,149,149,150,150,150,150,147,147,146,146,145,145,145,145,145,145,145,145,144,144,142,142,141,141,137,137,136,136,135,135,134,134,134,134,134,134,135,135,135,135,136,136,137,137,138,138,139,139,140,140,141,141,142,142,143,143,144,144,145,145,146,146,147,147,148,148,148,148,149,149,150,150,151,151,152,152,153,153,154,154,155,155,155,155,156,156,157,157,158,158,159,159,160,160,161,161,164,164,163,163,162,162,157,157,158,158,159,159,160,160,161,161,162,162,163,163,164,164,165,165,166,166,167,167,167,167,168,168,169,169,170,170,170,170,169,169,168,168,167,167,165,165,163,163,162,162,161,161,160,160,159,159,158,158,157,157,156,156,156,156,155,155,154,154,153,153,152,152,151,151,150,150,149,149,148,148,147,147,146,146,147,147,148,148,149,149,150,150,151,151,152,152,152,152,152,152,152,152,152,152,152,152,152,152,152,152,152,152,152,152,152,152,152,152,153,153,153,153,153,153,154,154,154,154,155,155,155,155,156,156,156,156,156,156,157,157,157,157,158,158,158,158,158,158,159,159,159,159,160,160,160,160,160,160,161,161,161,161,161,161,162,162,162,162,162,162,163,163,163,163,163,163,163,163,163,163,163,163,163,163,163,163,162,162,162,162,161,161,161,161,160,160,159,159,158,158,155,155,152,152,151,151,151,151,151,151,150,150,149,149,149,149,148,148,147,147,147,147,146,146,145,145,144,144,142,142,141,141,140,140,139,139,138,138,138,138,140,140,141,141,142,142,143,143,144,144,145,145,146,146,147,147,148,148,149,149,150,150,151,151,152,152,153,153,154,154,155,155,156,156,156,156,157,157,158,158,159,159,160,160,164,164,164,164,164,164,163,163,163,163,162,162,162,162,161,161,161,161,160,160,160,160,159,159,158,158,157,157,157,157,156,156,155,155,155,155,154,154,154,154,154,154,155,155,155,155,155,155,156,156,156,156,157,157,157,157,157,157,158,158,158,158,159,159,159,159,160,160,160,160,160,160,161,161,161,161,162,162,162,162,163,163,163,163,164,164,164,164,165,165,165,165,166,166,166,166,167,167,167,167,167,167,168,168,168,168,169,169,169,169,169,169,170,170,171,171,171,171,171,171,172,172,172,172,172,172,173,173,173,173,173,173,174,174,174,174,172,172,171,171,171,171,171,171,171,171,170,170,170,170,170,170,170,170,169,169,169,169,169,169,164,164,165,165,165,165,166,166,166,166,166,166,166,166,167,167,167,167,167,167,167,167,167,167,163,163,162,162,156,156,155,155,154,154,153,153,152,152,151,151,157,157,158,158,159,159,160,160,161,161,162,162,161,161,160,160,159,159,158,158,157,157,156,156,155,155,154,154,153,153,152,152,151,151,150,150,149,149,149,149,148,148,147,147,146,146,148,148,147,147,146,146,145,145,145,145,144,144,143,143,142,142,141,141,140,140,139,139,138,138,137,137,136,136,135,135,134,134,134,134,134,134,135,135,136,136,137,137,138,138,139,139,140,140,141,141,142,142,143,143,144,144,124,124,124,124,124,124,124,124,123,123,122,122,123,123,123,123,123,123,123,123,123,123,123,123,123,123,123,123,121,121,122,122,123,123,124,124,125,125,125,125,126,126,126,126,127,127,128,128,129,129,130,130,131,131,132,132,133,133,134,134,135,135,136,136,137,137,137,137,138,138,139,139,140,140,141,141,140,140,139,139,138,138,138,138,137,137,136,136,135,135,134,134,134,134,133,133,132,132,132,132,131,131,130,130,129,129,128,128,127,127,126,126,123,123,122,122,122,122,121,121,120,120,120,120,119,119,121,121,122,122,123,123,124,124,124,124,125,125,126,126,126,126,127,127,127,127,128,128,128,128,129,129,129,129,130,130,130,130,131,131,132,132,132,132,133,133,133,133,134,134,135,135,136,136,136,136,136,136,135,135,135,135,134,134,134,134,133,133,133,133,132,132,132,132,131,131,130,130,129,129,128,128,127,127,126,126,125,125,124,124,123,123,122,122,121,121,120,120,119,119,118,118,117,117,116,116,116,116,116,116,115,115,115,115,115,115,114,114,114,114,114,114,113,113,113,113,112,112,111,111,111,111,110,110,109,109,110,110,111,111,111,111,112,112,113,113,114,114,114,114,115,115,116,116,116,116,117,117,117,117,118,118,117,117,118,118,118,118,119,119,120,120,120,120,121,121,121,121,121,121,121,121,121,121,121,121,121,121,118,118,118,118,118,118,119,119,120,120,121,121,122,122,122,122,123,123,123,123,123,123,123,123,123,123,123,123,122,122,121,121,120,120,120,120,119,119,119,119,119,119,119,119,117,117,116,116,117,117,116,116,115,115,115,115,114,114,113,113,112,112,111,111,110,110,110,110,110,110,111,111,112,112,113,113,114,114,114,114,114,114,115,115,115,115,115,115,115,115,114,114,113,113,113,113,113,113,113,113,112,112,111,111,111,111,111,111,112,112,113,113,112,112,111,111,110,110,109,109,108,108,107,107,106,106,106,106,107,107,107,107,108,108,107,107,107,107,107,107,107,107,107,107,107,107,107,107,108,108,108,108,108,108,108,108,108,108,108,108,109,109,110,110,111,111,110,110,110,110,109,109,112,112,113,113,113,113,111,111,111,111,111,111,113,113,114,114,115,115,116,116,117,117,118,118,118,118,117,117,116,116,115,115,116,116,118,118,119,119,120,120,120,120,121,121,122,122,123,123,124,124,124,124,125,125,125,125,125,125,124,124,124,124,124,124,123,123,123,123,122,122,121,121,119,119,119,119,120,120,121,121,121,121,121,121,121,121,122,122,122,122,123,123,123,123,123,123,124,124,124,124,118,118,118,118,119,119,119,119,119,119,118,118,118,118,117,117,116,116,116,116,116,116,116,116,115,115,114,114,114,114,114,114,114,114,111,111,111,111,112,112,113,113,114,114,116,116,117,117,116,116,115,115,114,114,113,113,112,112,111,111,110,110,109,109,108,108,107,107,106,106,106,106,106,106,106,106,106,106,106,106,106,106,106,106,106,106,105,105,105,105,105,105,105,105,106,106,105,105,105,105,105,105,105,105,105,105,105,105,105,105,105,105,104,104,104,104,104,104,104,104,105,105,106,106,107,107,108,108,109,109,110,110,111,111,112,112,112,112,113,113,114,114,114,114,115,115,116,116,116,116,117,117,118,118,118,118,118,118,118,118,117,117,117,117,116,116,116,116,115,115,115,115,114,114,114,114,113,113,113,113,113,113,112,112,112,112,111,111,110,110,110,110,109,109,108,108,107,107,106,106,105,105,104,104,103,103,102,102,101,101,100,100,99,99,99,99,99,99,98,98,98,98,97,97,96,96,95,95,94,94,95,95,94,94,93,93,93,93,92,92,90,90,91,91,92,92,91,91,90,90,89,89,89,89,89,89,89,89,90,90,90,90,91,91,92,92,93,93,94,94,96,96,97,97,97,97,97,97,96,96,95,95,93,93,92,92,91,91,90,90,90,90,90,90,89,89,89,89,89,89,89,89,89,89,89,89,89,89,89,89,88,88,88,88,88,88,87,87,87,87,87,87,87,87,87,87,87,87,86,86,86,86,85,85,85,85,85,85,84,84,84,84,83,83,83,83,83,83,82,82,82,82,81,81,81,81,80,80,80,80,79,79,79,79,78,78,78,78,78,78,78,78,78,78,78,78,79,79,79,79,80,80,81,81,82,82,83,83,84,84,85,85,84,84,87,87,86,86,88,88,89,89,90,90,90,90,90,90,90,90,90,90,90,90,91,91,96,96,97,97,98,98,98,98,98,98,98,98,97,97,96,96,95,95,95,95,95,95,95,95,92,92,92,92,92,92,92,92,92,92,93,93,94,94,95,95,95,95,96,96,97,97,98,98,99,99,100,100,101,101,102,102,103,103,104,104,105,105,106,106,107,107,108,108,109,109,110,110,111,111,112,112,113,113,113,113,112,112,111,111,110,110,109,109,108,108,115,115,116,116,117,117,117,117,118,118,118,118,119,119,119,119,119,119,119,119,120,120,120,120,120,120,120,120,121,121,121,121,121,121,121,121,121,121,121,121,123,123,123,123,123,123,123,123,123,123,123,123,122,122,122,122,122,122,122,122,122,122,121,121,121,121,121,121,121,121,121,121,120,120,120,120,120,120,120,120,120,120,119,119,119,119,119,119,119,119,119,119,119,119,119,119,119,119,119,119,119,119,123,123,123,123,124,124,124,124,125,125,126,126,126,126,126,126,126,126,126,126,126,126,126,126,126,126,126,126,127,127,127,127,128,128,128,128,129,129,130,130,130,130,130,130,131,131,131,131,131,131,132,132,132,132,133,133,133,133,132,132,132,132,132,132,131,131,131,131,131,131,130,130,130,130,129,129,128,128,128,128,127,127,127,127,127,127,127,127,127,127,128,128,128,128,128,128,128,128,128,128,128,128,127,127,126,126,126,126,126,126,126,126,126,126,126,126,125,125,125,125,125,125,125,125,125,125,126,126,127,127,124,124,123,123,122,122,121,121,121,121,121,121,120,120,120,120,120,120,119,119,119,119,118,118,118,118,117,117,117,117,116,116,116,116,115,115,115,115,114,114,113,113,112,112,112,112,111,111,110,110,109,109,108,108,107,107,106,106,105,105,104,104,104,104,103,103,103,103,102,102,101,101,101,101,100,100,100,100,99,99,99,99,99,99,96,96,96,96,97,97,97,97,97,97,97,97,97,97,98,98,99,99,99,99,99,99,99,99,99,99,98,98,98,98,101,101,102,102,103,103,101,101,101,101,101,101,102,102,103,103,104,104,104,104,104,104,104,104,111,111,110,110,109,109,108,108,107,107,106,106,105,105,104,104,103,103,102,102,102,102,103,103,104,104,105,105,106,106,106,106,107,107,108,108,109,109,110,110,111,111,112,112,112,112,113,113,113,113,116,116,116,116,116,116,116,116,116,116,116,116,116,116,116,116,116,116,116,116,117,117,118,118,118,118,118,118,118,118,118,118,118,118,118,118,118,118,118,118,118,118,118,118,117,117,115,115,115,115,115,115,116,116,117,117,114,114,113,113,112,112,111,111,110,110,110,110,109,109,109,109,108,108,108,108,107,107,106,106,105,105,105,105,104,104,104,104,103,103,103,103,102,102,101,101,101,101,100,100,100,100,102,102,98,98,97,97,98,98,97,97,99,99,98,98,98,98,98,98,99,99,99,99,98,98,97,97,96,96,96,96,96,96,96,96,95,95,94,94,93,93,92,92,92,92,91,91,91,91,90,90,83,83,84,84,85,85,86,86,87,87,88,88,89,89,90,90,91,91,92,92,93,93,94,94,95,95,96,96,97,97,98,98,98,98,96,96,95,95,94,94,93,93,92,92,91,91,90,90,89,89,88,88,87,87,86,86,85,85,84,84,83,83,82,82,83,83,84,84,85,85,86,86,87,87,88,88,89,89,89,89,90,90,91,91,92,92,93,93,90,90,89,89,87,87,86,86,79,79,73,73,72,72,72,72,74,74,74,74,75,75,75,75,75,75,76,76,76,76,76,76,76,76,77,77,77,77,78,78,78,78,79,79,79,79,80,80,81,81,81,81,81,81,81,81,80,80,79,79,79,79,79,79,78,78,78,78,77,77,77,77,76,76,76,76,75,75,75,75,74,74,74,74,74,74,74,74,73,73,72,72,72,72,72,72,71,71,70,70,70,70,70,70,70,70,70,70,70,70,70,70,69,69,68,68,68,68,69,69,69,69,69,69,70,70,70,70,70,70,70,70,71,71,71,71,72,72,73,73,73,73,74,74,75,75,76,76,78,78,77,77,76,76,75,75,74,74,74,74,73,73,73,73,74,74,75,75,74,74,73,73,73,73,72,72,72,72,71,71,71,71,69,69,70,70,71,71,72,72,73,73,73,73,73,73,74,74,74,74,75,75,75,75,76,76,76,76,77,77,77,77,78,78,78,78,79,79,79,79,80,80,80,80,81,81,81,81,82,82,83,83,83,83,83,83,82,82,81,81,80,80,79,79,79,79,78,78,77,77,76,76,75,75,76,76,77,77,77,77,78,78,79,79,79,79,80,80,81,81,81,81,82,82,82,82,83,83,83,83,80,80,81,81,82,82,83,83,83,83,83,83,84,84,84,84,89,89,88,88,87,87,86,86,85,85,84,84,83,83,82,82,81,81,80,80,79,79,78,78,77,77,76,76,76,76,75,75,75,75,74,74,73,73,73,73,72,72,72,72,71,71,71,71,70,70,70,70,70,70,69,69,69,69,68,68,68,68,68,68,67,67,67,67,66,66,66,66,66,66,66,66,65,65,65,65,65,65,65,65,65,65,65,65,65,65,65,65,65,65,65,65,65,65,65,65,65,65,66,66,66,66,66,66,67,67,67,67,68,68,68,68,68,68,68,68,68,68,68,68,68,68,69,69,69,69,70,70,70,70,71,71,71,71,71,71,72,72,72,72,73,73,73,73,74,74,74,74,75,75,75,75,76,76,76,76,77,77,78,78,79,79,80,80,80,80,80,80,79,79,79,79,78,78,78,78,78,78,78,78,78,78,78,78,78,78,78,78,78,78,78,78,78,78,78,78,78,78,84,84,84,84,86,86,87,87,88,88,89,89,90,90,90,90,89,89,88,88,88,88,87,87,86,86,86,86,87,87,87,87,87,87,88,88,88,88,89,89,89,89,90,90,90,90,91,91,91,91,92,92,93,93,93,93,94,94,95,95,96,96,97,97,97,97,105,105,105,105,106,106,106,106,106,106,106,106,107,107,108,108,108,108,108,108,108,108,108,108,107,107,107,107,107,107,109,109,109,109,109,109,109,109,127,127,127,127,126,126,126,126,125,125,124,124,123,123,122,122,122,122,121,121,120,120,119,119,118,118,117,117,116,116,115,115,114,114,114,114,115,115,116,116,117,117,118,118,119,119,120,120,121,121,122,122,123,123,124,124,125,125,126,126,131,131,132,132,133,133,134,134,134,134,135,135,135,135,137,137,138,138,139,139,140,140,141,141,142,142,147,147,147,147,146,146,145,145,144,144,143,143,142,142,141,141,140,140,139,139,138,138,137,137,136,136,135,135,134,134,133,133,134,134,134,134,133,133,132,132,131,131,130,130,129,129,128,128,127,127,128,128,129,129,130,130,131,131,132,132,133,133,132,132,131,131,130,130,131,131,130,130,129,129,128,128,128,128,127,127,126,126,125,125,122,122,124,124,124,124,124,124,124,124,125,125,126,126,127,127,128,128,129,129,130,130,131,131,133,133,134,134,134,134,136,136,136,136,137,137,138,138,138,138,138,138,138,138,136,136,136,136,135,135,134,134,134,134,135,135,137,137,140,140,141,141,142,142,143,143,144,144,145,145,141,141,142,142,143,143,144,144,145,145,146,146,146,146,146,146,146,146,149,149,150,150,151,151,149,149,150,150,151,151,152,152,153,153,154,154,155,155,156,156,157,157,158,158,159,159,160,160,161,161,161,161,162,162,163,163,164,164,165,165,165,165,166,166,167,167,168,168,169,169,170,170,171,171,172,172,173,173,174,174,175,175,176,176,176,176,175,175,174,174,173,173,172,172,171,171,170,170,169,169,168,168,167,167,166,166,165,165,164,164,164,164,163,163,162,162,161,161,160,160,159,159,158,158,157,157,156,156,155,155,154,154,153,153,153,153,152,152,151,151,150,150,149,149,148,148,149,149,150,150,151,151,152,152,153,153,153,153,153,153,153,153,153,153,153,153,153,153,154,154,154,154,154,154,154,154,154,154,153,153,152,152,151,151,150,150,149,149,150,150,151,151,152,152,153,153,156,156,156,156,156,156,156,156,156,156,156,156,156,156,155,155,155,155,155,155,155,155,155,155,155,155,167,167,169,169,170,170,171,171,172,172,173,173,174,174,175,175,176,176,177,177,178,178,179,179,180,180,181,181,182,182,183,183,184,184,185,185,186,186,187,187,188,188,189,189,190,190,191,191,192,192,193,193,194,194,205,205,204,204,203,203,202,202,201,201,200,200,199,199,198,198,197,197,196,196,195,195,194,194,193,193,192,192,191,191,190,190,189,189,188,188,187,187,186,186,185,185,184,184,183,183,182,182,181,181,179,179,178,178,177,177,176,176,175,175,174,174,173,173,172,172,171,171,170,170,169,169,168,168,167,167,166,166,165,165,164,164,163,163,162,162,161,161,160,160,159,159,158,158,157,157,156,156,155,155,154,154,153,153,152,152,151,151,150,150,149,149,148,148,147,147,146,146,145,145,144,144,143,143,142,142,141,141,140,140,139,139,138,138,137,137,136,136,135,135,134,134,134,134,133,133,132,132,132,132,131,131,131,131,130,130,130,130,130,130,129,129,129,129,130,130,130,130,130,130,130,130,130,130,131,131,131,131,132,132,132,132,132,132,133,133,134,134,134,134,135,135,136,136,137,137,138,138,139,139,140,140,141,141,142,142,143,143,144,144,145,145,146,146,147,147,148,148,149,149,150,150,151,151,152,152,153,153,154,154,155,155,156,156,157,157,158,158,159,159,160,160,161,161,162,162,163,163,164,164,165,165,166,166,167,167,168,168,169,169,170,170,171,171,172,172,173,173,174,174,175,175,176,176,177,177,178,178,179,179,180,180,181,181,182,182,183,183,184,184,185,185,186,186,187,187,187,187,188,188,189,189,190,190,191,191,192,192,192,192,193,193,194,194,195,195,196,196,197,197,198,198,199,199,200,200,201,201,201,201,202,202,203,203,204,204,205,205,206,206,207,207,207,207,208,208,209,209,209,209,208,208,208,208,207,207,206,206,205,205,204,204,203,203,202,202,201,201,200,200,199,199,198,198,197,197,196,196,195,195,194,194,193,193,193,193,192,192,191,191,190,190,189,189,188,188,188,188,187,187,186,186,185,185,184,184,183,183,182,182,181,181,180,180,179,179,178,178,177,177,176,176,175,175,174,174,173,173,172,172,171,171,170,170,169,169,168,168,167,167,166,166,165,165,164,164,163,163,162,162,161,161,160,160,159,159,158,158,157,157,156,156,156,156,155,155,153,153,152,152,148,148,138,138,143,143,142,142,141,141,140,140,139,139,137,137,136,136,135,135,134,134,133,133,132,132,131,131,130,130,129,129,128,128,127,127,126,126,125,125,124,124,123,123,122,122,121,121,120,120,119,119,118,118,117,117,116,116,115,115,114,114,113,113,112,112,111,111,110,110,109,109,108,108,107,107,106,106,106,106,105,105,104,104,104,104,103,103,102,102,102,102,101,101,100,100,100,100,99,99,98,98,98,98,97,97,96,96,95,95,94,94,93,93,93,93,92,92,91,91,91,91,90,90,89,89,89,89,88,88,88,88,87,87,86,86,86,86,85,85,85,85,84,84,84,84,83,83,83,83,82,82,82,82,81,81,81,81,80,80,80,80,80,80,79,79,79,79,79,79,78,78,78,78,78,78,60,60,60,60,60,60,60,60,60,60,59,59,59,59,58,58,58,58,58,58,57,57,57,57,56,56,56,56,55,55,55,55,55,55,54,54,54,54,53,53,53,53,52,52,52,52,51,51,51,51,50,50,50,50,49,49,48,48,47,47,46,46,45,45,44,44,43,43,42,42,42,42,41,41,40,40,40,40,36,36,36,36,36,36,36,36,35,35,35,35,34,34,34,34,33,33,33,33,32,32,31,31,31,31,30,30,30,30,29,29,29,29,28,28,28,28,27,27,27,27,26,26,26,26,26,26,26,26,26,26,26,26,27,27,28,28,29,29,30,30,31,31,32,32,33,33,34,34,35,35,36,36,36,36,36,36,36,36,35,35,32,32,31,31,31,31,35,35,35,35,35,35,34,34,34,34,35,35,36,36,39,39,39,39,39,39,39,39,39,39,39,39,40,40,36,36,35,35,34,34,33,33,32,32,31,31,30,30,29,29,28,28,27,27,26,26,26,26,26,26,26,26,26,26,26,26,27,27,28,28,29,29,32,32,33,33,34,34,36,36,36,36,36,36,36,36,35,35,33,33,34,34,35,35,35,35,30,30,29,29,28,28,27,27,26,26,26,26,26,26,26,26,26,26,27,27,28,28,29,29,30,30,31,31,32,32,32,32,31,31,30,30,29,29,28,28,27,27,26,26,26,26,26,26,26,26,26,26,26,26,27,27,27,27,28,28,29,29,29,29,30,30,28,28,27,27,26,26,26,26,26,26,26,26,26,26,27,27,28,28,29,29,30,30,31,31,31,31,30,30,29,29,28,28,27,27,26,26,26,26,26,26,26,26,26,26,27,27,28,28,29,29,31,31,30,30,30,30,31,31,31,31,30,30,30,30,29,29,28,28,28,28,27,27,27,27,28,28,29,29,28,28,27,27,26,26,26,26,26,26,26,26,25,25,27,27,26,26,26,26,26,26,26,26,26,26,26,26,26,26,26,26,26,26,27,27,29,29,28,28,27,27,26,26,26,26,26,26,26,26,26,26,26,26,26,26,26,26,26,26,26,26,30,30,30,30,29,29,30,30,31,31,32,32,33,33,34,34,33,33,33,33,33,33,34,34,33,33,33,33,32,32,31,31,31,31,30,30,30,30,29,29,28,28,27,27,27,27,27,27,27,27,26,26,26,26,26,26,26,26,26,26,26,26,26,26,26,26,26,26,27,27,26,26,28,28,28,28,28,28,29,29,28,28,28,28,28,28,30,30,30,30,29,29,29,29,28,28,28,28,27,27,27,27,26,26,26,26,26,26,26,26,25,25,26,26,27,27,28,28,29,29,30,30,31,31,32,32,33,33,34,34,35,35,36,36,36,36,36,36,36,36,36,36,35,35,35,35,34,34,34,34,34,34,35,35,36,36,36,36,35,35,32,32,32,32,31,31,31,31,31,31,31,31,31,31,32,32,32,32,33,33,34,34,35,35,37,37,37,37,37,37,37,37,36,36,36,36,36,36,36,36,36,36,35,35,34,34,33,33,32,32,31,31,31,31,30,30,30,30,30,30,30,30,28,28,29,29,30,30,31,31,31,31,32,32,32,32,32,32,32,32,33,33,34,34,34,34,34,34,36,36,37,37,36,36,36,36,34,34,33,33,34,34,34,34,34,34,35,35,36,36,36,36,34,34,35,35,36,36,37,37,36,36,36,36,35,35,35,35,34,34,35,35,36,36,36,36,37,37,36,36,36,36,35,35,33,33,34,34,34,34,35,35,36,36,36,36,36,36,36,36,34,34,34,34,34,34,34,34,33,33,36,36,36,36,36,36,36,36,36,36,36,36,36,36,35,35,34,34,33,33,32,32,32,32,32,32,32,32,32,32,32,32,32,32,31,31,30,30,30,30,30,30,29,29,30,30,30,30,29,29,28,28,28,28,28,28,28,28,28,28,28,28,28,28,29,29,30,30,31,31,32,32,32,32,33,33,33,33,34,34,35,35,35,35,36,36,36,36,37,37,37,37,37,37,36,36,36,36,35,35,34,34,33,33,32,32,31,31,30,30,31,31,30,30,29,29,28,28,27,27,26,26,26,26,26,26,26,26,26,26,26,26,27,27,28,28,29,29,30,30,31,31,32,32,33,33,32,32,33,33,34,34,34,34,35,35,36,36,36,36,37,37,36,36,36,36,35,35,33,33,32,32,30,30,34,34,35,35,36,36,36,36,36,36,36,36,36,36,36,36,35,35,35,35,34,34,33,33,32,32,33,33,34,34,35,35,36,36,37,37,37,37,36,36,36,36,35,35,34,34,33,33,33,33,34,34,35,35,36,36,36,36,36,36,36,36,36,36,36,36,39,39,39,39,39,39,39,39,40,40,40,40,40,40,41,41,41,41,42,42,42,42,41,41,41,41,43,43,43,43,41,41,41,41,41,41,41,41,41,41,42,42,42,42,43,43,44,44,45,45,46,46,50,50,52,52,53,53,54,54,55,55,56,56,56,56,56,56,57,57,55,55,59,59,59,59,58,58,58,58,57,57,57,57,57,57,56,56,56,56,55,55,55,55,54,54,54,54,53,53,53,53,52,52,52,52,51,51,50,50,51,51,52,52,53,53,44,44,44,44,42,42,42,42,43,43,43,43,42,42,41,41,41,41,41,41,41,41,41,41,43,43,43,43,46,46,44,44,43,43,42,42,42,42,39,39,39,39,40,40,40,40,41,41,41,41,42,42,42,42,43,43,44,44,45,45,46,46,47,47,48,48,49,49,50,50,50,50,51,51,50,50,50,50,49,49,49,49,48,48,48,48,47,47,47,47,46,46,46,46,46,46,46,46,46,46,47,47,48,48,49,49,50,50,51,51,52,52,52,52,51,51,50,50,50,50,51,51,52,52,51,51,51,51,52,52,52,52,53,53,54,54,54,54,54,54,54,54,54,54,54,54,55,55,56,56,56,56,56,56,56,56,55,55,54,54,54,54,49,49,48,48,47,47,46,46,46,46,46,46,47,47,47,47,48,48,48,48,47,47,46,46,46,46,46,46,46,46,47,47,48,48,49,49,49,49,49,49,49,49,50,50,50,50,51,51,52,52,53,53,54,54,55,55,56,56,56,56,56,56,56,56,56,56,56,56,55,55,54,54,53,53,52,52,52,52,51,51,51,51,50,50,50,50,49,49,49,49,48,48,48,48,47,47,47,47,46,46,46,46,46,46,46,46,46,46,46,46,46,46,47,47,48,48,49,49,49,49,49,49,49,49,49,49,49,49,50,50,52,52,52,52,52,52,52,52,52,52,51,51,53,53,54,54,54,54,54,54,54,54,54,54,54,54,53,53,48,48,49,49,50,50,51,51,52,52,53,53,54,54,55,55,56,56,56,56,56,56,56,56,56,56,56,56,56,56,56,56,56,56,56,56,56,56,55,55,55,55,57,57,55,55,54,54,54,54,53,53,53,53,52,52,52,52,51,51,50,50,50,50,49,49,49,49,48,48,48,48,47,47,47,47,46,46,46,46,46,46,46,46,47,47,48,48,49,49,50,50,51,51,52,52,51,51,51,51,51,51,52,52,53,53,56,56,56,56,56,56,56,56,56,56,55,55,55,55,55,55,56,56,56,56,56,56,56,56,56,56,56,56,55,55,54,54,53,53,52,52,55,55,56,56,56,56,56,56,56,56,56,56,55,55,54,54,53,53,54,54,53,53,52,52,51,51,50,50,49,49,48,48,47,47,47,47,46,46,46,46,46,46,46,46,46,46,46,46,46,46,49,49,49,49,49,49,53,53,54,54,55,55,56,56,56,56,56,56,56,56,56,56,55,55,54,54,54,54,53,53,52,52,52,52,52,52,51,51,50,50,49,49,48,48,48,48,46,46,47,47,47,47,47,47,47,47,46,46,46,46,46,46,46,46,46,46,46,46,46,46,46,46,49,49,49,49,50,50,50,50,48,48,48,48,49,49,50,50,51,51,51,51,52,52,52,52,52,52,53,53,54,54,54,54,54,54,54,54,54,54,54,54,55,55,56,56,57,57,57,57,57,57,57,57,57,57,57,57,57,57,57,57,56,56,56,56,55,55,55,55,54,54,53,53,52,52,52,52,51,51,51,51,51,51,49,49,49,49,49,49,48,48,48,48,49,49,49,49,50,50,51,51,51,51,52,52,52,52,53,53,53,53,54,54,54,54,55,55,55,55,55,55,56,56,56,56,57,57,57,57,58,58,58,58,59,59,59,59,59,59,60,60,60,60,61,61,61,61,61,61,61,61,60,60,60,60,59,59,59,59,59,59,58,58,58,58,57,57,57,57,56,56,56,56,56,56,55,55,55,55,54,54,54,54,53,53,53,53,52,52,51,51,52,52,53,53,54,54,55,55,56,56,57,57,57,57,56,56,57,57,56,56,55,55,55,55,55,55,54,54,54,54,53,53,52,52,44,44,43,43,42,42,41,41,41,41,41,41,41,41,41,41,43,43,42,42,43,43,44,44,45,45,46,46,48,48,50,50,52,52,51,51,51,51,50,50,49,49,47,47,46,46,45,45,44,44,43,43,42,42,42,42,41,41,40,40,40,40,39,39,39,39,39,39,39,39,39,39,39,39,39,39,39,39,40,40,40,40,41,41,41,41,42,42,42,42,42,42,42,42,43,43,43,43,43,43,41,41,41,41,41,41,41,41,41,41,42,42,42,42,43,43,47,47,48,48,47,47,46,46,45,45,44,44,43,43,42,42,42,42,41,41,40,40,40,40,39,39,39,39,39,39,39,39,39,39,39,39,39,39,40,40,41,41,41,41,36,36,35,35,35,35,36,36,36,36,36,36,36,36,35,35,34,34,33,33,33,33,33,33,34,34,35,35,36,36,36,36,36,36,37,37,36,36,35,35,34,34,33,33,32,32,31,31,30,30,29,29,28,28,27,27,26,26,26,26,26,26,26,26,26,26,26,26,29,29,30,30,30,30,26,26,26,26,26,26,26,26,27,27,27,27,28,28,30,30,31,31,34,34,33,33,33,33,32,32,31,31,30,30,29,29,28,28,27,27,26,26,26,26,26,26,26,26,26,26,26,26,27,27,27,27,26,26,26,26,26,26,26,26,27,27,28,28,28,28,28,28,28,28,29,29,29,29,30,30,31,31,31,31,32,32,33,33,34,34,35,35,36,36,36,36,36,36,36,36,36,36,35,35,34,34,33,33,32,32,31,31,31,31,31,31,30,30,30,30,29,29,29,29,28,28,28,28,27,27,27,27,25];
	VAR num array_z{8510}:= [0,0,0,0,0,0,0,0,0,0,0,0,0,0,0,0,0,0,0,0,0,0,0,0,0,0,0,0,0,0,-5,-5,0,0,0,0,0,0,0,0,0,0,0,0,0,0,0,0,0,0,0,0,0,0,0,0,0,0,0,0,0,0,0,0,0,0,0,0,0,0,0,0,0,0,0,0,0,0,0,0,0,0,0,0,0,0,0,0,0,0,0,0,0,0,0,0,0,0,0,0,0,0,0,0,0,0,0,0,0,0,0,0,0,0,0,0,0,0,0,0,0,0,0,0,0,0,0,0,0,0,0,0,0,0,0,0,0,0,0,0,0,0,0,0,0,0,0,0,0,0,0,0,0,0,0,0,0,0,0,0,0,0,0,0,0,0,0,0,0,0,0,0,0,0,0,0,0,0,0,0,0,0,0,0,0,0,0,0,0,0,0,0,0,0,0,0,0,0,0,0,0,0,0,0,0,0,0,0,0,0,0,0,0,0,0,0,0,0,0,0,0,0,0,0,0,0,0,0,0,0,0,0,0,0,0,0,0,0,0,0,0,0,0,0,0,0,0,0,0,0,0,0,0,0,0,0,0,0,0,0,0,0,0,0,0,0,0,0,0,0,0,0,-5,-5,0,0,0,0,0,0,0,0,0,0,0,0,0,0,0,0,0,0,0,0,0,0,0,0,0,0,0,0,0,0,0,0,0,0,0,0,0,0,0,0,0,0,0,0,0,0,0,0,0,0,0,0,0,0,0,0,0,0,0,0,0,0,0,0,0,0,0,0,0,0,0,0,0,0,0,0,0,0,0,0,0,0,0,0,0,0,0,0,0,0,0,0,0,0,0,0,0,0,0,0,0,0,0,0,0,0,0,0,0,0,0,0,0,0,0,0,0,0,0,0,0,0,0,0,0,0,0,0,0,0,0,0,-5,-5,0,0,0,0,0,0,0,0,0,0,0,0,0,0,-5,-5,0,0,0,0,0,0,0,0,0,0,0,0,0,0,0,0,-5,-5,0,0,0,0,0,0,0,0,0,0,0,0,0,0,0,0,0,0,0,0,0,0,0,0,0,0,-5,-5,-5,-5,-5,-5,0,0,0,0,-5,-5,-5,-5,-5,-5,0,0,0,0,0,0,0,0,0,0,0,0,0,0,0,0,0,0,0,0,0,0,0,0,0,0,0,0,0,0,0,0,-5,-5,0,0,0,0,0,0,0,0,0,0,0,0,0,0,0,0,0,0,0,0,-5,-5,-5,-5,0,0,0,0,0,0,-5,-5,-5,-5,0,0,-5,-5,0,0,0,0,0,0,0,0,0,0,0,0,0,0,0,0,0,0,0,0,0,0,0,0,0,0,0,0,0,0,0,0,0,0,0,0,0,0,0,0,0,0,0,0,0,0,0,0,0,0,0,0,0,0,0,0,0,0,0,0,0,0,0,0,0,0,0,0,-5,-5,0,0,0,0,0,0,0,0,0,0,0,0,0,0,0,0,0,0,0,0,0,0,0,0,0,0,0,0,0,0,0,0,0,0,0,0,0,0,0,0,0,0,0,0,0,0,0,0,0,0,0,0,0,0,0,0,0,0,0,0,0,0,0,0,0,0,0,0,0,0,0,0,-5,-5,0,0,0,0,0,0,0,0,0,0,0,0,0,0,-5,-5,0,0,0,0,0,0,0,0,0,0,0,0,0,0,0,0,0,0,0,0,0,0,0,0,0,0,0,0,0,0,0,0,-5,-5,-5,-5,-5,-5,-5,-5,0,0,0,0,0,0,0,0,0,0,0,0,0,0,0,0,0,0,0,0,0,0,0,0,0,0,0,0,0,0,0,0,0,0,0,0,0,0,-5,-5,0,0,0,0,0,0,0,0,-5,-5,-5,-5,-5,-5,-5,-5,0,0,0,0,0,0,0,0,0,0,0,0,0,0,0,0,0,0,0,0,0,0,0,0,0,0,0,0,0,0,0,0,0,0,0,0,0,0,0,0,0,0,0,0,0,0,0,0,0,0,0,0,0,0,0,0,0,0,0,0,0,0,0,0,0,0,0,0,0,0,0,0,0,0,0,0,0,0,0,0,0,0,0,0,0,0,0,0,0,0,0,0,0,0,0,0,0,0,0,0,0,0,0,0,0,0,0,0,0,0,0,0,0,0,0,0,0,0,0,0,0,0,-5,-5,0,0,0,0,0,0,0,0,0,0,0,0,0,0,0,0,-5,-5,0,0,0,0,0,0,0,0,0,0,0,0,0,0,0,0,0,0,0,0,0,0,0,0,0,0,0,0,0,0,-5,-5,0,0,0,0,-5,-5,0,0,0,0,0,0,0,0,0,0,-5,-5,0,0,0,0,0,0,0,0,0,0,0,0,-5,-5,0,0,0,0,0,0,-5,-5,0,0,0,0,0,0,0,0,0,0,0,0,-5,-5,0,0,0,0,0,0,0,0,0,0,0,0,0,0,-5,-5,0,0,0,0,0,0,0,0,0,0,0,0,0,0,0,0,0,0,0,0,0,0,0,0,0,0,0,0,0,0,0,0,0,0,0,0,0,0,0,0,0,0,-5,-5,0,0,0,0,0,0,0,0,0,0,0,0,0,0,0,0,0,0,0,0,0,0,0,0,0,0,0,0,0,0,0,0,0,0,0,0,0,0,0,0,0,0,0,0,0,0,0,0,0,0,0,0,0,0,0,0,-5,-5,0,0,0,0,0,0,0,0,0,0,0,0,0,0,0,0,0,0,0,0,0,0,0,0,0,0,0,0,0,0,0,0,0,0,0,0,0,0,0,0,0,0,0,0,0,0,0,0,0,0,0,0,-5,-5,0,0,0,0,0,0,0,0,0,0,0,0,0,0,0,0,0,0,0,0,0,0,0,0,0,0,0,0,0,0,0,0,0,0,0,0,-5,-5,0,0,0,0,0,0,0,0,0,0,0,0,0,0,0,0,0,0,-5,-5,-5,-5,0,0,0,0,0,0,0,0,0,0,0,0,0,0,0,0,0,0,0,0,0,0,0,0,0,0,0,0,0,0,0,0,0,0,0,0,0,0,0,0,0,0,0,0,0,0,0,0,0,0,0,0,0,0,0,0,0,0,0,0,-5,-5,0,0,0,0,0,0,0,0,0,0,0,0,0,0,0,0,0,0,0,0,0,0,0,0,0,0,-5,-5,0,0,0,0,0,0,0,0,-5,-5,0,0,0,0,0,0,0,0,-5,-5,0,0,0,0,0,0,0,0,0,0,0,0,0,0,0,0,0,0,0,0,0,0,0,0,0,0,0,0,0,0,0,0,0,0,-5,-5,0,0,0,0,0,0,0,0,0,0,0,0,0,0,0,0,0,0,0,0,0,0,0,0,0,0,0,0,0,0,0,0,0,0,0,0,0,0,0,0,0,0,0,0,0,0,-5,-5,0,0,0,0,0,0,0,0,0,0,0,0,0,0,0,0,0,0,0,0,0,0,0,0,0,0,0,0,0,0,0,0,0,0,-5,-5,0,0,0,0,0,0,-5,-5,0,0,0,0,0,0,0,0,0,0,0,0,0,0,0,0,0,0,0,0,0,0,0,0,0,0,0,0,0,0,0,0,-5,-5,0,0,0,0,0,0,0,0,0,0,-5,-5,0,0,0,0,0,0,-5,-5,0,0,0,0,0,0,0,0,0,0,-5,-5,0,0,0,0,0,0,0,0,-5,-5,0,0,0,0,0,0,0,0,0,0,0,0,-5,-5,0,0,0,0,0,0,0,0,0,0,0,0,0,0,0,0,0,0,0,0,-5,-5,0,0,0,0,-5,-5,0,0,0,0,0,0,0,0,0,0,0,0,-5,-5,0,0,0,0,0,0,0,0,0,0,0,0,0,0,0,0,-5,-5,0,0,0,0,0,0,-5,-5,0,0,0,0,0,0,0,0,0,0,0,0,0,0,0,0,0,0,0,0,0,0,0,0,0,0,0,0,0,0,0,0,0,0,0,0,0,0,0,0,0,0,0,0,0,0,0,0,0,0,0,0,0,0,0,0,0,0,0,0,0,0,0,0,0,0,0,0,0,0,0,0,0,0,-5,-5,0,0,0,0,0,0,0,0,-5,-5,0,0,0,0,0,0,0,0,0,0,0,0,0,0,0,0,0,0,0,0,0,0,-5,-5,0,0,0,0,0,0,0,0,0,0,0,0,0,0,0,0,0,0,0,0,0,0,0,0,0,0,0,0,0,0,-5,-5,-5,-5,0,0,0,0,0,0,0,0,0,0,0,0,0,0,0,0,-5,-5,0,0,0,0,0,0,0,0,0,0,0,0,0,0,0,0,0,0,0,0,0,0,0,0,0,0,0,0,0,0,0,0,0,0,0,0,0,0,0,0,0,0,0,0,0,0,0,0,0,0,0,0,0,0,0,0,0,0,0,0,0,0,0,0,0,0,0,0,0,0,0,0,0,0,0,0,0,0,0,0,0,0,0,0,0,0,0,0,0,0,0,0,0,0,0,0,0,0,0,0,0,0,0,0,0,0,0,0,0,0,0,0,0,0,0,0,0,0,-5,-5,0,0,0,0,0,0,0,0,0,0,0,0,0,0,0,0,0,0,0,0,0,0,0,0,0,0,0,0,0,0,0,0,0,0,0,0,0,0,0,0,0,0,0,0,0,0,0,0,0,0,0,0,0,0,-5,-5,-5,-5,-5,-5,0,0,0,0,0,0,0,0,-5,-5,0,0,-5,-5,0,0,0,0,0,0,0,0,0,0,0,0,0,0,0,0,0,0,0,0,0,0,0,0,0,0,0,0,0,0,0,0,0,0,0,0,0,0,0,0,0,0,0,0,0,0,0,0,0,0,0,0,0,0,0,0,0,0,0,0,0,0,0,0,0,0,0,0,0,0,-5,-5,0,0,0,0,-5,-5,0,0,0,0,0,0,0,0,0,0,0,0,0,0,0,0,0,0,0,0,0,0,0,0,0,0,0,0,0,0,0,0,0,0,0,0,-5,-5,-5,-5,0,0,0,0,0,0,0,0,0,0,0,0,0,0,0,0,0,0,0,0,0,0,0,0,0,0,0,0,0,0,0,0,0,0,0,0,-5,-5,0,0,0,0,0,0,0,0,0,0,0,0,0,0,0,0,0,0,0,0,0,0,0,0,0,0,0,0,0,0,0,0,0,0,0,0,0,0,0,0,0,0,0,0,0,0,0,0,0,0,0,0,0,0,0,0,0,0,0,0,0,0,0,0,0,0,0,0,0,0,0,0,0,0,0,0,0,0,0,0,0,0,0,0,0,0,0,0,0,0,0,0,0,0,0,0,0,0,0,0,0,0,0,0,0,0,0,0,0,0,0,0,0,0,-5,-5,-5,-5,0,0,0,0,0,0,0,0,0,0,0,0,0,0,0,0,0,0,0,0,0,0,0,0,-5,-5,0,0,0,0,0,0,0,0,0,0,-5,-5,0,0,0,0,0,0,0,0,0,0,0,0,0,0,-5,-5,0,0,-5,-5,0,0,0,0,0,0,0,0,0,0,0,0,0,0,0,0,0,0,0,0,0,0,-5,-5,0,0,0,0,0,0,0,0,0,0,0,0,0,0,0,0,0,0,0,0,0,0,0,0,0,0,0,0,0,0,0,0,0,0,0,0,0,0,0,0,0,0,0,0,0,0,0,0,0,0,0,0,0,0,0,0,0,0,0,0,0,0,0,0,0,0,0,0,0,0,0,0,0,0,0,0,0,0,0,0,0,0,0,0,0,0,0,0,0,0,0,0,0,0,0,0,0,0,0,0,0,0,0,0,0,0,0,0,0,0,0,0,0,0,0,0,0,0,0,0,0,0,0,0,0,0,0,0,0,0,0,0,0,0,0,0,0,0,0,0,0,0,0,0,0,0,0,0,0,0,0,0,-5,-5,0,0,0,0,-5,-5,0,0,0,0,0,0,0,0,0,0,0,0,0,0,0,0,0,0,0,0,0,0,-5,-5,0,0,-5,-5,0,0,0,0,0,0,0,0,0,0,-5,-5,0,0,0,0,0,0,0,0,0,0,0,0,0,0,0,0,0,0,0,0,0,0,0,0,0,0,0,0,0,0,0,0,0,0,0,0,0,0,0,0,0,0,0,0,-5,-5,0,0,0,0,0,0,0,0,0,0,0,0,0,0,0,0,0,0,0,0,0,0,0,0,0,0,0,0,0,0,0,0,0,0,0,0,0,0,0,0,0,0,0,0,0,0,0,0,0,0,0,0,0,0,-5,-5,0,0,0,0,0,0,0,0,0,0,0,0,0,0,0,0,0,0,0,0,0,0,0,0,0,0,-5,-5,0,0,0,0,-5,-5,0,0,0,0,0,0,0,0,0,0,0,0,0,0,0,0,0,0,0,0,0,0,0,0,0,0,0,0,0,0,0,0,0,0,0,0,0,0,0,0,-5,-5,0,0,0,0,0,0,0,0,0,0,0,0,0,0,0,0,0,0,0,0,0,0,0,0,0,0,0,0,0,0,0,0,0,0,-5,-5,0,0,0,0,0,0,0,0,0,0,0,0,0,0,0,0,0,0,0,0,0,0,0,0,0,0,0,0,0,0,0,0,0,0,0,0,0,0,0,0,0,0,0,0,0,0,0,0,0,0,0,0,0,0,0,0,0,0,0,0,0,0,0,0,0,0,0,0,0,0,0,0,0,0,0,0,0,0,0,0,0,0,0,0,0,0,0,0,0,0,0,0,0,0,0,0,0,0,0,0,0,0,0,0,0,0,0,0,0,0,0,0,0,0,0,0,0,0,0,0,0,0,0,0,0,0,0,0,0,0,0,0,0,0,0,0,0,0,0,0,0,0,0,0,0,0,0,0,0,0,0,0,0,0,0,0,0,0,0,0,0,0,0,0,0,0,0,0,-5,-5,0,0,0,0,0,0,0,0,0,0,0,0,0,0,0,0,0,0,0,0,0,0,-5,-5,-5,-5,0,0,0,0,0,0,0,0,0,0,0,0,0,0,0,0,0,0,0,0,0,0,0,0,0,0,0,0,0,0,0,0,0,0,0,0,0,0,0,0,0,0,-5,-5,0,0,-5,-5,0,0,0,0,0,0,-5,-5,0,0,-5,-5,0,0,0,0,0,0,0,0,0,0,0,0,0,0,0,0,0,0,0,0,0,0,0,0,0,0,0,0,0,0,0,0,0,0,0,0,0,0,0,0,0,0,0,0,0,0,-5,-5,0,0,0,0,-5,-5,0,0,-5,-5,0,0,0,0,0,0,0,0,0,0,0,0,0,0,0,0,0,0,0,0,0,0,-5,-5,0,0,0,0,-5,-5,0,0,0,0,0,0,0,0,0,0,0,0,0,0,-5,-5,0,0,0,0,0,0,-5,-5,0,0,0,0,0,0,0,0,0,0,-5,-5,0,0,0,0,0,0,0,0,0,0,0,0,0,0,0,0,0,0,0,0,0,0,0,0,-5,-5,0,0,0,0,0,0,0,0,0,0,0,0,0,0,0,0,0,0,0,0,0,0,0,0,0,0,0,0,0,0,0,0,-5,-5,0,0,0,0,0,0,0,0,0,0,0,0,0,0,0,0,0,0,0,0,0,0,0,0,0,0,-5,-5,0,0,0,0,0,0,0,0,0,0,0,0,0,0,0,0,0,0,0,0,0,0,0,0,0,0,0,0,0,0,0,0,-5,-5,0,0,0,0,0,0,0,0,-5,-5,0,0,0,0,0,0,0,0,0,0,0,0,0,0,0,0,0,0,0,0,0,0,0,0,0,0,0,0,0,0,0,0,0,0,0,0,0,0,0,0,0,0,0,0,0,0,0,0,0,0,0,0,0,0,0,0,0,0,0,0,0,0,0,0,0,0,0,0,0,0,0,0,0,0,0,0,0,0,0,0,0,0,0,0,0,0,0,0,0,0,0,0,0,0,0,0,0,0,0,0,0,0,0,0,0,0,0,0,0,0,0,0,0,0,0,0,0,0,0,0,0,0,0,0,0,0,0,0,0,0,0,0,0,0,0,0,0,0,0,0,0,0,0,0,0,0,0,0,0,0,0,0,0,0,0,0,0,0,0,0,0,0,0,0,0,0,0,0,0,0,0,0,0,0,0,0,0,0,0,0,0,0,0,0,-5,-5,0,0,0,0,0,0,0,0,-5,-5,0,0,0,0,0,0,0,0,0,0,0,0,0,0,0,0,0,0,0,0,0,0,0,0,0,0,0,0,-5,-5,0,0,0,0,0,0,0,0,0,0,-5,-5,0,0,0,0,0,0,0,0,0,0,0,0,0,0,0,0,0,0,0,0,0,0,0,0,0,0,0,0,0,0,0,0,0,0,0,0,0,0,0,0,0,0,0,0,0,0,0,0,0,0,0,0,0,0,0,0,0,0,0,0,0,0,0,0,0,0,0,0,0,0,0,0,0,0,0,0,0,0,0,0,0,0,0,0,0,0,0,0,0,0,0,0,0,0,0,0,0,0,0,0,0,0,0,0,-5,-5,-5,-5,0,0,-5,-5,0,0,0,0,0,0,0,0,0,0,0,0,0,0,0,0,0,0,0,0,-5,-5,0,0,0,0,0,0,0,0,0,0,0,0,0,0,0,0,0,0,0,0,0,0,-5,-5,0,0,0,0,0,0,0,0,0,0,0,0,0,0,0,0,0,0,0,0,0,0,0,0,0,0,0,0,0,0,0,0,0,0,0,0,0,0,0,0,0,0,0,0,0,0,0,0,0,0,0,0,0,0,-5,-5,0,0,0,0,0,0,0,0,-5,-5,0,0,0,0,0,0,0,0,0,0,0,0,0,0,0,0,0,0,0,0,0,0,0,0,0,0,-5,-5,0,0,0,0,0,0,0,0,0,0,0,0,0,0,0,0,0,0,0,0,0,0,0,0,0,0,0,0,0,0,0,0,0,0,0,0,0,0,0,0,0,0,0,0,0,0,0,0,0,0,0,0,0,0,0,0,0,0,0,0,0,0,0,0,0,0,0,0,0,0,0,0,-5,-5,0,0,0,0,0,0,0,0,0,0,0,0,0,0,0,0,0,0,0,0,0,0,0,0,0,0,0,0,0,0,0,0,0,0,0,0,0,0,0,0,0,0,0,0,0,0,0,0,0,0,0,0,0,0,0,0,0,0,0,0,0,0,0,0,0,0,0,0,0,0,0,0,0,0,0,0,0,0,0,0,0,0,0,0,0,0,0,0,0,0,0,0,0,0,0,0,0,0,0,0,0,0,0,0,0,0,0,0,0,0,0,0,0,0,0,0,0,0,0,0,0,0,0,0,0,0,-5,-5,-5,-5,0,0,0,0,0,0,0,0,0,0,0,0,0,0,0,0,0,0,0,0,0,0,0,0,0,0,0,0,0,0,0,0,0,0,0,0,0,0,0,0,0,0,0,0,-5,-5,0,0,0,0,0,0,0,0,0,0,0,0,0,0,0,0,0,0,0,0,0,0,0,0,0,0,0,0,0,0,0,0,0,0,0,0,-5,-5,0,0,0,0,0,0,0,0,0,0,0,0,0,0,0,0,0,0,0,0,0,0,0,0,0,0,0,0,-5,-5,0,0,0,0,-5,-5,0,0,0,0,0,0,0,0,0,0,0,0,0,0,0,0,-5,-5,0,0,0,0,0,0,0,0,0,0,0,0,0,0,0,0,0,0,0,0,0,0,0,0,0,0,0,0,0,0,0,0,0,0,0,0,0,0,0,0,0,0,0,0,0,0,0,0,-5,-5,0,0,0,0,0,0,0,0,0,0,0,0,0,0,0,0,0,0,0,0,0,0,0,0,0,0,0,0,0,0,0,0,0,0,0,0,0,0,0,0,0,0,0,0,-5,-5,0,0,0,0,0,0,0,0,-5,-5,0,0,0,0,0,0,0,0,0,0,0,0,0,0,0,0,0,0,0,0,0,0,0,0,0,0,0,0,0,0,0,0,0,0,0,0,0,0,0,0,0,0,0,0,-5,-5,-5,-5,0,0,-5,-5,0,0,0,0,0,0,0,0,0,0,0,0,0,0,0,0,0,0,-5,-5,0,0,0,0,0,0,0,0,0,0,0,0,0,0,0,0,0,0,0,0,0,0,-5,-5,0,0,0,0,0,0,0,0,0,0,0,0,0,0,0,0,0,0,0,0,0,0,0,0,0,0,0,0,0,0,0,0,0,0,0,0,0,0,0,0,0,0,0,0,0,0,0,0,0,0,0,0,0,0,0,0,0,0,0,0,0,0,-5,-5,0,0,0,0,0,0,0,0,0,0,0,0,0,0,0,0,0,0,0,0,0,0,-5,-5,0,0,-5,-5,0,0,-5,-5,-5,-5,-5,-5,0,0,-5,-5,0,0,0,0,0,0,0,0,0,0,0,0,0,0,0,0,0,0,0,0,0,0,0,0,0,0,0,0,0,0,0,0,0,0,0,0,0,0,0,0,0,0,0,0,0,0,0,0,0,0,0,0,0,0,0,0,0,0,0,0,0,0,0,0,0,0,0,0,0,0,-5,-5,0,0,0,0,0,0,0,0,0,0,0,0,0,0,0,0,0,0,0,0,0,0,0,0,0,0,0,0,0,0,0,0,0,0,0,0,0,0,0,0,0,0,0,0,0,0,0,0,0,0,0,0,0,0,0,0,-5,-5,-5,-5,0,0,0,0,-5,-5,0,0,-5,-5,0,0,0,0,0,0,0,0,-5,-5,-5,-5,0,0,0,0,0,0,-5,-5,0,0,-5,-5,0,0,0,0,-5,-5,0,0,0,0,0,0,0,0,0,0,0,0,0,0,0,0,0,0,0,0,0,0,0,0,0,0,0,0,0,0,0,0,0,0,0,0,0,0,0,0,0,0,0,0,0,0,0,0,0,0,0,0,0,0,0,0,0,0,0,0,0,0,-5,-5,0,0,0,0,0,0,0,0,0,0,0,0,0,0,0,0,0,0,0,0,0,0,0,0,0,0,-5,-5,0,0,0,0,0,0,0,0,0,0,0,0,0,0,-5,-5,0,0,0,0,0,0,0,0,0,0,0,0,0,0,0,0,0,0,0,0,0,0,0,0,0,0,0,0,0,0,0,0,0,0,0,0,0,0,0,0,0,0,0,0,0,0,0,0,0,0,0,0,0,0,0,0,0,0,0,0,0,0,0,0,0,0,0,0,0,0,0,0,0,0,0,0,0,0,0,0,0,0,0,0,0,0,0,0,0,0,0,0,0,0,0,0,0,0,0,0,0,0,0,0,0,0,0,0,0,0,0,0,0,0,0,0,0,0,0,0,0,0,0,0,0,0,0,0,0,0,0,0,0,0,0,0,0,0,0,0,0,0,0,0,0,0,0,0,0,0,0,0,0,0,0,0,0,0,0,0,0,0,0,0,0,0,0,0,0,0,0,0,0,0,0,0,0,0,0,0,0,0,0,0,0,0,0,0,0,0,0,0,0,0,0,0,0,0,0,0,-5,-5,0,0,-5,-5,-5,-5,-5,-5,0,0,0,0,0,0,0,0,0,0,0,0,0,0,-5,-5,0,0,0,0,0,0,0,0,0,0,0,0,0,0,0,0,0,0,0,0,0,0,0,0,0,0,0,0,0,0,0,0,0,0,0,0,0,0,-5,-5,-5,-5,0,0,-5,-5,0,0,0,0,0,0,-5,-5,0,0,0,0,0,0,0,0,0,0,-5,-5,0,0,0,0,0,0,0,0,0,0,0,0,-5,-5,0,0,0,0,0,0,0,0,0,0,0,0,0,0,0,0,0,0,0,0,0,0,0,0,0,0,0,0,0,0,0,0,0,0,0,0,0,0,0,0,0,0,0,0,0,0,0,0,0,0,0,0,0,0,0,0,0,0,-5,-5,0,0,0,0,0,0,0,0,0,0,0,0,0,0,0,0,0,0,0,0,0,0,0,0,-5,-5,0,0,0,0,0,0,0,0,0,0,-5,-5,0,0,0,0,0,0,0,0,0,0,0,0,0,0,0,0,0,0,0,0,0,0,0,0,0,0,0,0,0,0,0,0,0,0,0,0,0,0,0,0,0,0,0,0,0,0,0,0,0,0,0,0,0,0,-5,-5,0,0,0,0,0,0,0,0,0,0,0,0,0,0,-5,-5,0,0,0,0,0,0,0,0,0,0,0,0,0,0,0,0,0,0,0,0,0,0,-5,-5,0,0,0,0,-5,-5,0,0,0,0,0,0,0,0,0,0,0,0,-5,-5,0,0,0,0,0,0,0,0,0,0,-5,-5,-5,-5,0,0,0,0,0,0,0,0,0,0,-5,-5,0,0,0,0,0,0,0,0,0,0,0,0,0,0,0,0,-5,-5,0,0,0,0,-5,-5,0,0,0,0,0,0,0,0,0,0,0,0,0,0,0,0,0,0,0,0,0,0,0,0,0,0,0,0,0,0,0,0,0,0,0,0,0,0,0,0,0,0,0,0,0,0,0,0,0,0,0,0,0,0,0,0,0,0,0,0,0,0,0,0,0,0,0,0,0,0,0,0,0,0,0,0,0,0,0,0,0,0,0,0,0,0,0,0,0,0,0,0,0,0,0,0,0,0,0,0,0,0,0,0,0,0,0,0,0,0,0,0,0,0,0,0,0,0,-5,-5,0,0,0,0,0,0,0,0,0,0,0,0,0,0,0,0,0,0,0,0,0,0,0,0,0,0,0,0,0,0,0,0,0,0,0,0,0,0,0,0,0,0,-5,-5,0,0,0,0,0,0,-5,-5,0,0,0,0,0,0,0,0,0,0,0,0,0,0,0,0,0,0,0,0,0,0,0,0,-5,-5,-5,-5,0,0,0,0,0,0,0,0,0,0,0,0,0,0,0,0,0,0,0,0,0,0,0,0,0,0,0,0,0,0,0,0,0,0,0,0,0,0,0,0,0,0,0,0,0,0,0,0,0,0,-5,-5,0,0,0,0,0,0,0,0,0,0,0,0,0,0,0,0,0,0,0,0,0,0,0,0,0,0,0,0,0,0,0,0,0,0,0,0,0,0,0,0,0,0,0,0,0,0,0,0,-5,-5,0,0,0,0,0,0,0,0,0,0,0,0,0,0,0,0,0,0,0,0,-5,-5,0,0,0,0,0,0,0,0,0,0,0,0,0,0,0,0,0,0,0,0,0,0,0,0,0,0,0,0,0,0,0,0,0,0,0,0,0,0,0,0,0,0,0,0,0,0,0,0,0,0,0,0,0,0,0,0,0,0,0,0,0,0,0,0,0,0,0,0,0,0,0,0,0,0,0,0,0,0,0,0,0,0,0,0,0,0,0,0,0,0,0,0,0,0,0,0,0,0,0,0,0,0,0,0,0,0,0,0,0,0,0,0,0,0,0,0,0,0,0,0,0,0,0,0,0,0,0,0,0,0,0,0,0,0,0,0,0,0,0,0,0,0,0,0,0,0,0,0,0,0,0,0,0,0,0,0,0,0,0,0,0,0,0,0,0,0,0,0,0,0,0,0,0,0,0,0,0,0,0,0,0,0,0,0,0,0,0,0,0,0,0,0,0,0,0,0,0,0,0,0,0,0,0,0,0,0,0,0,0,0,0,0,0,0,0,0,0,0,0,0,0,0,0,0,0,0,0,0,0,0,0,0,0,0,0,0,0,0,0,0,0,0,0,0,0,0,0,0,0,0,0,0,0,0,0,0,0,0,0,0,0,0,0,0,0,0,0,0,0,0,0,0,0,0,0,0,0,0,0,0,0,0,0,0,0,0,0,0,0,0,0,0,0,0,0,0,0,0,0,0,0,0,0,0,0,0,0,0,0,0,0,0,0,0,0,0,0,0,0,0,0,0,0,0,0,0,0,0,0,0,0,0,0,0,0,0,0,0,0,0,0,0,0,0,0,0,0,0,0,0,0,0,0,0,0,0,0,0,0,0,0,0,0,0,0,0,0,0,0,0,0,0,0,0,0,0,0,0,0,0,0,0,0,0,0,0,0,0,0,0,0,0,-5,-5,-5,-5,-5,-5,-5,-5,-5,-5,0,0,0,0,0,0,0,0,-5,-5,0,0,0,0,0,0,0,0,0,0,0,0,0,0,0,0,0,0,0,0,0,0,0,0,0,0,0,0,0,0,0,0,0,0,0,0,0,0,0,0,0,0,0,0,0,0,0,0,0,0,0,0,0,0,0,0,0,0,0,0,0,0,0,0,0,0,0,0,0,0,0,0,0,0,0,0,0,0,0,0,0,0,0,0,0,0,0,0,0,0,0,0,0,0,0,0,0,0,0,0,0,0,0,0,0,0,0,0,0,0,0,0,0,0,0,0,0,0,0,0,0,0,0,0,0,0,0,0,0,0,0,0,0,0,0,0,0,0,0,0,0,0,0,0,0,0,0,0,0,0,0,0,0,0,0,0,0,0,0,0,-5,-5,0,0,0,0,0,0,0,0,0,0,0,0,0,0,0,0,0,0,0,0,0,0,0,0,0,0,0,0,0,0,0,0,0,0,0,0,0,0,0,0,0,0,0,0,0,0,0,0,0,0,0,0,0,0,0,0,0,0,0,0,0,0,0,0,0,0,0,0,0,0,0,0,0,0,0,0,-5,-5,0,0,0,0,0,0,-5,-5,0,0,0,0,0,0,0,0,0,0,0,0,0,0,0,0,0,0,0,0,0,0,0,0,0,0,0,0,0,0,0,0,0,0,0,0,0,0,0,0,0,0,0,0,0,0,0,0,0,0,0,0,0,0,0,0,0,0,0,0,0,0,0,0,0,0,0,0,0,0,0,0,-5,-5,0,0,0,0,-5,-5,0,0,0,0,0,0,0,0,0,0,0,0,-5,-5,0,0,0,0,0,0,0,0,0,0,0,0,-5,-5,0,0,0,0,0,0,0,0,0,0,0,0,0,0,0,0,0,0,0,0,0,0,0,0,0,0,0,0,0,0,0,0,0,0,0,0,-5,-5,0,0,0,0,-5,-5,0,0,0,0,0,0,0,0,-5,-5,0,0,0,0,0,0,-5,-5,0,0,0,0,0,0,0,0,0,0,0,0,0,0,0,0,0,0,0,0,0,0,0,0,0,0,0,0,-5,-5,0,0,0,0,0,0,0,0,0,0,0,0,0,0,0,0,0,0,0,0,0,0,0,0,0,0,0,0,0,0,0,0,0,0,-5,-5,0,0,0,0,0,0,0,0,0,0,0,0,0,0,0,0,0,0,0,0,0,0,0,0,0,0,0,0,0,0,0,0,0,0,0,0,0,0,0,0,0,0,0,0,0,0,0,0,-5,-5,0,0,0,0,-5,-5,0,0,0,0,0,0,0,0,0,0,0,0,0,0,-5,-5,0,0,0,0,0,0,0,0,0,0,0,0,0,0,0,0,-5,-5,-5,-5,0,0,0,0,0,0,0,0,0,0,0,0,0,0,0,0,0,0,0,0,-5,-5,0,0,0,0,0,0,0,0,0,0,0,0,0,0,0,0,0,0,0,0,0,0,0,0,-5,-5,0,0,0,0,-5,-5,0,0,0,0,0,0,0,0,-5,-5,0,0,0,0,0,0,-5,-5,0,0,0,0,0,0,0,0,0,0,0,0,0,0,0,0,0,0,0,0,-5,-5,0,0,0,0,0,0,0,0,0,0,0,0,0,0,0,0,0,0,0,0,0,0,0,0,-5,-5,0,0,0,0,0,0,-5,-5,0,0,0,0,-5,-5,0,0,0,0,0,0,0,0,0,0,0,0,0,0,0,0,0,0,0,0,0,0,0,0,0,0,0,0,0,0,0,0,0,0,0,0,0,0,0,0,0,0,0,0,0,0,0,0,0,0,0,0,0,0,0,0,0,0,0,0,0,0,0,0,0,0,-5,-5,0,0,0,0,-5,-5,0,0,0,0,0,0,0,0,-5,-5,0,0,0,0,0,0,0,0,0,0,0,0,-5,-5,0,0,0,0,0,0,-5,-5,0,0,0,0,0,0,0,0,-5,-5,0,0,0,0,0,0,0,0,0,0,0,0,0,0,0,0,0,0,-5,-5,0,0,0,0,0,0,0,0,0,0,0,0,0,0,0,0,0,0,0,0,0,0,0,0,0,0,0,0,0,0,0,0,-5,-5,0,0,0,0,0,0,0,0,0,0,0,0,0,0,-5,-5,0,0,0,0,0,0,0,0,0,0,0,0,0,0,-5,-5,0,0,0,0,0,0,0,0,0,0,0,0,0,0,-5,-5,0,0,0,0,0,0,0,0,0,0,0,0,0,0,-5,-5,0,0,0,0,0,0,0,0,-5,-5,0,0,0,0,0,0,0,0,0,0,0,0,0,0,0,0,0,0,0,0,-5,-5,0,0,0,0,0,0,0,0,0,0,0,0,-5,-5,0,0,0,0,0,0,-5,-5,0,0,0,0,0,0,0,0,0,0,0,0,0,0,0,0,-5,-5,0,0,0,0,0,0,-5,-5,0,0,0,0,0,0,0,0,0,0,0,0,0,0,0,0,0,0,0,0,0,0,0,0,0,0,0,0,0,0,0,0,0,0,0,0,0,0,-5,-5,0,0,0,0,0,0,0,0,0,0,0,0,0,0,0,0,0,0,0,0,0,0,0,0,0,0,-5,-5,0,0,0,0,0,0,-5,-5,0,0,0,0,-5,-5,0,0,0,0,0,0,0,0,0,0,0,0,0,0,-5,-5,0,0,-5,-5,-5,-5,0,0,0,0,0,0,0,0,0,0,0,0,0,0,0,0,0,0,0,0,0,0,-5,-5,0,0,0,0,0,0,0,0,0,0,0,0,0,0,0,0,0,0,0,0,0,0,0,0,0,0,0,0,0,0,0,0,0,0,0,0,0,0,0,0,-5,-5,0,0,0,0,0,0,0,0,0,0,0,0,0,0,0,0,-5,-5,0,0,0,0,0,0,-5,-5,0,0,-5,-5,0,0,0,0,0,0,0,0,0,0,0,0,0,0,0,0,0,0,0,0,-5,-5,-5,-5,0,0,0,0,-5,-5,0,0,0,0,0,0,0,0,-5,-5,-5,-5,0,0,0,0,0,0,0,0,0,0,0,0,0,0,0,0,0,0,0,0,0,0,0,0,0,0,0,0,0,0,0,0,0,0,-5,-5,0,0,0,0,0,0,-5,-5,0,0,-5,-5,0,0,0,0,-5,-5,0,0,0,0,0,0,0,0,0,0,0,0,-5,-5,0,0,-5,-5,0,0,0,0,0,0,0,0,-5,-5,0,0,0,0,0,0,0,0,0,0,0,0,0,0,0,0,0,0,0,0,0,0,0,0,0,0,0,0,0,0,0,0,0,0,-5,-5,0,0,0,0,0,0,0,0,0,0,0,0,0,0,0,0,0,0,0,0,0,0,0,0,0,0,0,0,0,0,0,0,0,0,0,0,-5,-5,0,0,0,0,0,0,0,0,0,0,-5,-5,0,0,0,0,0,0,0,0,0,0,0,0,0,0,0,0,0,0,0,0,0,0,0,0,0,0,0,0,0,0,0,0,0,0,0,0,-5,-5,0,0,0,0,0,0,0,0,0,0,0,0,0,0,0,0,0,0,0,0,-5,-5,0,0,0,0,0,0,-5,-5,0,0,0,0,0,0,0,0,-5,-5,0,0,0,0,0,0,0,0,0,0,0,0,0,0,0,0,0,0,0,0,0,0,0,0,0,0,0,0,0,0,0,0,0,0,0,0,0,0,0,0,0,0,0,0,0,0,0,0,0,0,0,0,-5,-5,0,0,0,0,0,0,0,0,0,0,0,0,0,0,0,0,0,0,0,0,0,0,0,0,0,0,0,0,0,0,0,0,0,0,0,0,0,0,0,0,0,0,0,0,0,0,0,0,0,0,0,0,0,0,0,0,0,0,0,0,0,0,-5,-5,0,0,0,0,0,0,0,0,0,0,0,0,0,0,0,0,0,0,0,0,0,0,0,0,0,0,0,0,0,0,0,0,0,0,0,0,0,0,0,0,0,0,-5,-5,0,0,0,0,0,0,0,0,0,0,0,0,0,0,0,0,0,0,0,0,0,0,0,0,0,0,0,0,0,0,0,0,0,0,0,0,0,0,0,0,0,0,0,0,0,0,0,0,-5,-5,0,0,0,0,0,0,0,0,0,0,-5,-5,0,0,0,0,0,0,0,0,0,0,0,0,0,0,0,0,0,0,0,0,0,0,0,0,0,0,0,0,0,0,0,0,0,0,-5,-5,0,0,0,0,0,0,0,0,0,0,0,0,0,0,0,0,-5,-5,0,0,0,0,0,0,0,0,0,0,0,0,0,0,0,0,0,0,0,0,0,0,0,0,0,0,0,0,0,0,-5,-5,0,0,0,0,-5,-5,0,0,0,0,0,0,0,0,0,0,0,0,0,0,0,0,0,0,0,0,0,0,0,0,0,0,0,0,0,0,0,0,0,0,0,0,0,0,-5,-5,0,0,0,0,-5,-5,0,0,0,0,0,0,0,0,0,0,0,0,0,0,0,0,0,0,-5,-5,0,0,0,0,0,0,-5,-5,0,0,0,0,0,0,0,0,0,0,0,0,0,0,0,0,0,0,0,0,0,0,0,0,0,0,0,0,0,0,0,0,0,0,0,0,0,0,0,0,0,0,0,0,0,0,0,0,0,0,0,0,0,0,0,0,0,0,0,0,0,0,0,0,0,0,0,0,0,0,0,0,-5,-5,0,0,0,0,0,0,0,0,-5,-5,0,0,0,0,0,0,0,0,0,0,0,0,0,0,0,0,0,0,0,0,0,0,0,0,0,0,0,0,0,0,0,0,0,0,0,0,0,0,0,0,0,0,0,0,0,0,0,0,0,0,0,0,0,0,0,0,0,0,0,0,0,0,0,0,0,0,0,0,0,0,0,0,0,0,0,0,0,0,0,0,0,0,0,0,0,0,0,0,0,0,0,0,0,0,-5,-5,0,0,-5,-5,0,0,0,0,0,0,0,0,0,0,0,0,0,0,0,0,0,0,0,0,0,0,0,0,0,0,0,0,0,0,-5,-5,0,0,-5,-5,0,0,0,0,0,0,0,0,0,0,0,0,-5,-5,0,0,0,0,0,0,0,0,-5,-5,-5,-5,-5,-5,0,0,0,0,0,0,0,0,-5,-5,0,0,0,0,0,0,0,0,0,0,0,0,0,0,0,0,0,0,0,0,0,0,0,0,0,0,0,0,0,0,0,0,0,0,0,0,0,0,0,0,0,0,0,0,0,0,0,0,0,0,0,0,0,0,0,0,-5,-5,0,0,0,0,0,0,0,0,0,0,0,0,0,0,-5,-5,-5,-5,0,0,0,0,0,0,0,0,0,0,0,0,0,0,0,0,0,0,0,0,0,0,0,0,0,0,0,0,0,0,0,0,0,0,0,0,0,0,0,0,-5,-5,0,0,0,0,0,0,0,0,0,0,0,0,0,0,0,0,0,0,0,0,0,0,0,0,0,0,0,0,0,0,0,0,0,0,0,0,0,0,0,0,0,0,0,0,0,0,0,0,0,0,0,0,0,0,0,0,0,0,0,0,0,0,0,0,0,0,-5,-5,0,0,0,0,-5,-5,0,0,0,0,0,0,0,0,0,0,0,0,-5,-5,0,0,-5,-5,0,0,0,0,0,0,0,0,-5,-5,0,0,-5,-5,0,0,0,0,0,0,0,0,0,0,0,0,0,0,0,0,-5,-5,0,0,0,0,0,0,0,0,-5,-5,0,0,0,0,0,0,-5,-5,0,0,0,0,0,0,0,0,0,0,0,0,0,0,0,0,0,0,0,0,0,0,0,0,0,0,0,0,0,0,0,0,0,0,0,0,0,0,0,0,0,0,0,0,0,0,0,0,0,0,0,0,0,0,0,0,0,0,0,0];
	PROC main()
		MoveL home_1,v800,z100,pen\WObj:=paper_obj;
		FOR i FROM 1 TO Dim(array_x,1) DO
			MoveL Offs (origin,array_x{i},array_y{i},array_z{i}),v200,fine,pen\WObj:=paper_obj;
		ENDFOR
		MoveL home_1,v800,z100,pen\WObj:=paper_obj;
	ENDPROC
ENDMODULE
